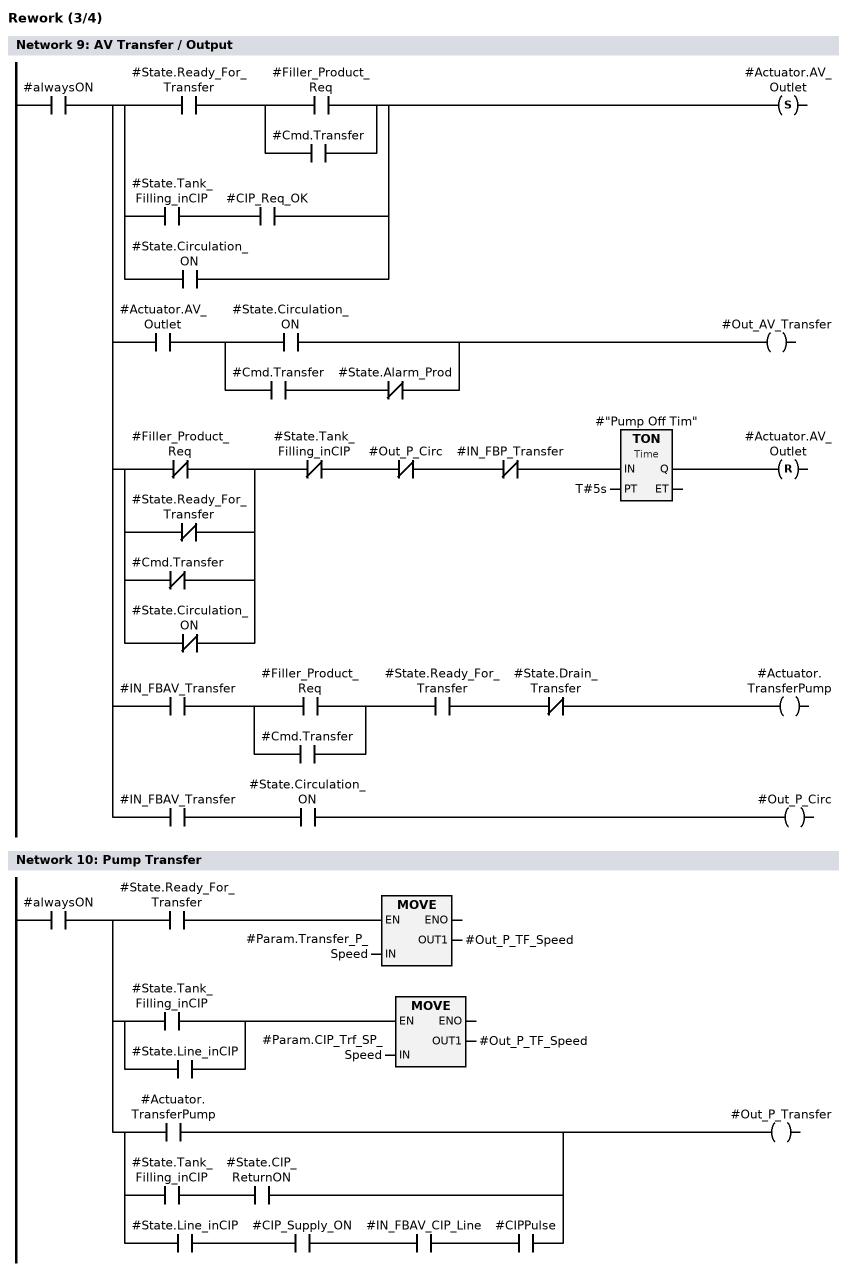
   RUNG wire#powerrail
      Contact( #alwaysON )
      wire#w1
      Contact( #State.Ready_For_Transfer )
      wire#w2
      Contact( #Filler_Product_Req )
      wire#w3
      S_Coil( #Actuator.AV_Outlet )
   END_RUNG
   RUNG wire#w2
      Contact( #Cmd.Transfer )
   END_RUNG wire#w3
   RUNG wire#w1
      Contact( #State.Tank_Filling_inCIP )
      Contact( #CIP_Req_OK )
   END_RUNG wire#w3
   RUNG wire#w1
      Contact( #State.Circulation_ON )
   END_RUNG wire#w3
   RUNG wire#w1
      Contact( #Actuator.AV_Outlet )
      wire#w4
      Contact( #State.Circulation_ON )
      wire#w5
      Coil( #Out_AV_Transfer )
   END_RUNG
   RUNG wire#w4
      Contact( #Cmd.Transfer )
      I_Contact( #State.Alarm_Prod )
   END_RUNG wire#w5
   RUNG wire#w1
      I_Contact( #Filler_Product_Req )
      wire#w6
      I_Contact( #State.Tank_Filling_inCIP )
      I_Contact( #Out_P_Circ )
      I_Contact( #IN_FBP_Transfer )
      { S7_Templates := "time_type := Time" } #"Pump Off Tim".TON(pt := T#5s, et =>)
      R_Coil( #Actuator.AV_Outlet )
   END_RUNG
   RUNG wire#w1
      I_Contact( #State.Ready_For_Transfer )
   END_RUNG wire#w6
   RUNG wire#w1
      I_Contact( #Cmd.Transfer )
   END_RUNG wire#w6
   RUNG wire#w1
      I_Contact( #State.Circulation_ON )
   END_RUNG wire#w6
   RUNG wire#w1
      Contact( #IN_FBAV_Transfer )
      wire#w7
      Contact( #Filler_Product_Req )
      wire#w8
      Contact( #State.Ready_For_Transfer )
      I_Contact( #State.Drain_Transfer )
      Coil( #Actuator.TransferPump )
   END_RUNG
   RUNG wire#w7
      Contact( #Cmd.Transfer )
   END_RUNG wire#w8
   RUNG wire#w1
      Contact( #IN_FBAV_Transfer )
      Contact( #State.Circulation_ON )
      Coil( #Out_P_Circ )
   END_RUNG
   // the same network as SCL:
   IF #alwaysON AND ((#State.Ready_For_Transfer AND (#Filler_Product_Req OR #Cmd.Transfer)) OR (#State.Tank_Filling_inCIP AND #CIP_Req_OK) OR #State.Circulation_ON) THEN
       #Actuator.AV_Outlet := TRUE;
   END_IF;
   #Out_AV_Transfer := #alwaysON AND #Actuator.AV_Outlet AND (#State.Circulation_ON OR (#Cmd.Transfer AND NOT #State.Alarm_Prod));
   #"Pump Off Tim"(IN := #alwaysON AND (NOT #Filler_Product_Req OR NOT #State.Ready_For_Transfer OR NOT #Cmd.Transfer OR NOT #State.Circulation_ON) AND NOT #State.Tank_Filling_inCIP AND NOT #Out_P_Circ AND NOT #IN_FBP_Transfer,   // TON
                   PT := T#5s);
   IF #"Pump Off Tim".Q THEN #Actuator.AV_Outlet := FALSE; END_IF;
   #Actuator.TransferPump := #alwaysON AND #IN_FBAV_Transfer AND (#Filler_Product_Req OR #Cmd.Transfer) AND #State.Ready_For_Transfer AND NOT #State.Drain_Transfer;
   #Out_P_Circ := #alwaysON AND #IN_FBAV_Transfer AND #State.Circulation_ON;
END_REGION

REGION Network 10: Pump Transfer
   RUNG wire#powerrail
      Contact( #alwaysON )
      wire#w1
      Contact( #State.Ready_For_Transfer )
      Move(in := #Param.Transfer_P_Speed, out1 => #Out_P_TF_Speed)
   END_RUNG
   RUNG wire#w1
      Contact( #State.Tank_Filling_inCIP )
      wire#w2
      Move(in := #Param.CIP_Trf_SP_Speed, out1 => #Out_P_TF_Speed)
   END_RUNG
   RUNG wire#w1
      Contact( #State.Line_inCIP )
   END_RUNG wire#w2
   RUNG wire#w1
      Contact( #Actuator.TransferPump )
      wire#w3
      Coil( #Out_P_Transfer )
   END_RUNG
   RUNG wire#w1
      Contact( #State.Tank_Filling_inCIP )
      Contact( #State.CIP_ReturnON )
   END_RUNG wire#w3
   RUNG wire#w1
      Contact( #State.Line_inCIP )
      Contact( #CIP_Supply_ON )
      Contact( #IN_FBAV_CIP_Line )
      Contact( #CIPPulse )
   END_RUNG wire#w3
   // the same network as SCL:
   IF #alwaysON AND #State.Ready_For_Transfer THEN #Out_P_TF_Speed := #Param.Transfer_P_Speed; END_IF;
   IF #alwaysON AND (#State.Tank_Filling_inCIP OR #State.Line_inCIP) THEN
       #Out_P_TF_Speed := #Param.CIP_Trf_SP_Speed;
   END_IF;
   #Out_P_Transfer := #alwaysON AND (#Actuator.TransferPump OR (#State.Tank_Filling_inCIP AND #State.CIP_ReturnON) OR (#State.Line_inCIP AND #CIP_Supply_ON AND #IN_FBAV_CIP_Line AND #CIPPulse));
END_REGION

REGION Network 11: State Transfer to FIlling
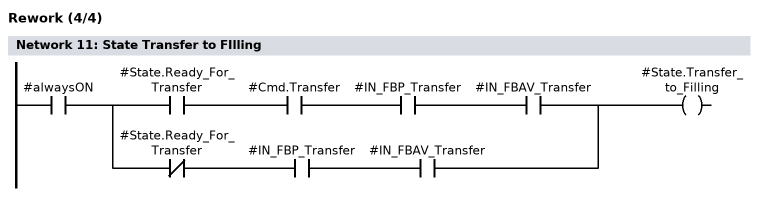
   RUNG wire#powerrail
      Contact( #alwaysON )
      wire#w1
      Contact( #State.Ready_For_Transfer )
      Contact( #Cmd.Transfer )
      Contact( #IN_FBP_Transfer )
      Contact( #IN_FBAV_Transfer )
      wire#w2
      Coil( #State.Transfer_to_Filling )
   END_RUNG
   RUNG wire#w1
      I_Contact( #State.Ready_For_Transfer )
      Contact( #IN_FBP_Transfer )
      Contact( #IN_FBAV_Transfer )
   END_RUNG wire#w2
   // the same network as SCL:
   #State.Transfer_to_Filling := #alwaysON AND ((#State.Ready_For_Transfer AND #Cmd.Transfer AND #IN_FBP_Transfer AND #IN_FBAV_Transfer) OR (NOT #State.Ready_For_Transfer AND #IN_FBP_Transfer AND #IN_FBAV_Transfer));
END_REGION
END_FUNCTION_BLOCK

FUNCTION_BLOCK "BFT_Type1"   // FB351, LAD
{ S7_Optimized_Access := 'TRUE' }
VERSION : 0.1
// Buffer Tank
// stored: AutoNumber false, IsIECCheckEnabled false, IsRetainMemResEnabled false, MemoryReserve 100, SetENOAutomatically false, UDAEnableTagReadback false
   VAR_INPUT
      "IN_FBAV.01" : Bool := FALSE;   // Tank Flushing Water Valve
      "IN_FBAV.02" : Bool := FALSE;   // Tank CIP Top Inlet Valve
      "IN_FBAV.03" : Bool := FALSE;   // Tank Tank Outlet Valve
      "IN_FBAV.04" : Bool := FALSE;   // Tank CIP Return Valve
      "IN_FBAV.05" : Bool := FALSE;   // Line CIP Bypass Valve
      "IN_FBAV.06" : Bool := FALSE;   // Tank Inlet Valve
      "IN_FBAV.07" : Bool := FALSE;   // Tank CIP Valve
      "IN_FBAV.08" : Bool := FALSE;   // Tank CIP Valve
      "IN_FBAV.09" : Bool := FALSE;   // Line CIP Valve
      IN_LT01 : Real;   // Tank Level Transmitter
      "IN_FBP.01" : Bool := FALSE;   // Transfer Pump
      "IN_P.01-Speed" : Real;   // Transfer Pump AV Speed
      "IN_FBP.02" : Bool := FALSE;   // CIP Pump
      "IN_P.02-Speed" : Real;   // CIP Pump AV Speed
      "IN_FBP.03" : Bool := FALSE;   // Supply Pump
      "IN_P.03-Speed" : Real;   // Supply Pump AV Speed
      DosePumpSpeed : Real;
      "DoseON-OFF" : Bool := FALSE;
      "DosePumpON-OFF" : Bool := FALSE;
      CIPPulse : Bool := FALSE;
      CIP_Supply_ON : Bool;
      LineTrf_OK : Bool := FALSE;
      LineFlush_OK : Bool;
      Loading_Busy : Bool;   // Other tank at loading
   END_VAR
   VAR_OUTPUT
      "OUT_AV.01" : Bool := FALSE;   // Tank Flushing Water Valve
      "OUT_AV.02" : Bool := FALSE;   // Tank CIP Top Inlet Valve
      "OUT_AV.03" : Bool := FALSE;   // Tank Tank Outlet Valve
      "OUT_AV.04" : Bool := FALSE;   // Tank CIP Return Valve
      "OUT_AV.05" : Bool := FALSE;   // Line CIP Bypass Valve
      "OUT_AV.06" : Bool := FALSE;   // Tank Inlet Valve
      "OUT_AV.07" : Bool := FALSE;   // Tank CIP Valve
      "OUT_AV.08" : Bool := FALSE;   // Tank CIP Valve
      "OUT_AV.09" : Bool := FALSE;   // Line CIP Valve
      "OUT_P.01" : Bool := FALSE;   // Transfer Pump
      "OUT_P.01-Speed" : Real;   // Transfer Pump AV Speed
      "OUT_P.02" : Bool := FALSE;   // CIP Pump
      "OUT_P.02-Speed" : Real;   // CIP Pump AV Speed
      "OUT_P.03" : Bool := FALSE;   // Supply Pump
      "OUT_P.03-Speed" : Real;   // Supply Pump AV Speed
      OUT_CIPTank_AVOpen : Bool;
      OUT_CIPLine_AVOpen : Bool;
   END_VAR
   VAR
      Cmd : Struct
         Inload : Bool;   // Start Loading
         Tank_CIP_Req : Bool;
         Line_CIP_Req : Bool;
         Flushing : Bool;   // Water Flushing
         RaadyForMix : Bool;   // Tank Ready for Blending
         Flush_Select : Byte;
      END_STRUCT;
      Param : Struct
         SP_Level_LL : Real := 10.0;
         SP_Level_ML : Real := 80.0;
         SP_Level_HL : Real := 100.0;
         SupplyPump_SP_Speed : Real := 80.0;
         L_Hi_Lim : Real := 100.0;
         L_Lo_Lim : Real := 0.0;
         L_Hys : Real := 5.0;
         FlushingTime : DInt := 10000;
         CIP_Trf_SP_Speed : Real := 80.0;
         CIP_Ret_ON_SP : Real := 5.0;
         CIP_Ret_OFF_SP : Real;
      END_STRUCT;
      State : Struct   // Tank in loading state
         Tank_inloading : Bool;
         Tank_inCIP : Bool;
         Line_inCIP : Bool;
         Flushing : Bool;
         Tank_LL : Bool;
         Tank_ML : Bool;
         Tank_HL : Bool;
         Inload_Enable : Bool;
         Tank_CIP_Enable : Bool;
         Line_CIP_Enable : Bool;
         Flushing_Enable : Bool;
         Flush_selected : Byte;
         CIP_Request_OK : Bool;
         CIP_ReturnON : Bool;
         Ready_For_Transfer_EN : Bool;   // Tank Ready for Transfer to Blending
         Ready_For_Transfer : Bool;   // Tank Ready for Transfer to Blending
         HWT_Status : Int;
         Transfer_to_Blend : Bool;
      END_STRUCT;
      alwaysON : Bool;
      L_Hys_Abs : Real;
      Hys_Level_HL : Real;
      Hys_Level_ML : Real;
      Hys_Level_LL : Real;
      r : Struct
         PosE1 : Bool;
         PosE2 : Bool;
         PosE3 : Bool;
         PosE4 : Bool;
         PosE5 : Bool;
         PosE6 : Bool;
         PosE7 : Bool;
         PosE8 : Bool;
         PosE9 : Bool;
         PosE10 : Bool;
         PosE11 : Bool;
         PosE12 : Bool;
         PosE13 : Bool;
         PosE14 : Bool;
         PosE15 : Bool;
         PosE16 : Bool;
         PosE17 : Bool;
         PosE18 : Bool;
         PosE19 : Bool;
         PosE20 : Bool;
         PosE21 : Bool;
         PosE22 : Bool;
         PosE23 : Bool;
         PosE24 : Bool;
         PosE25 : Bool;
         PosE26 : Bool;
         PosE27 : Bool;
         PosE28 : Bool;
         PosE29 : Bool;
         PosE30 : Bool;
         PosE31 : Bool;
         PosE32 : Bool;
      END_STRUCT;
      Actuator : Struct
         AV_Outlet : Bool;
         TransferPump : Bool;
         FlushPump : Bool;
         CV_Steam : Bool;
         Pump : Bool;
      END_STRUCT;
      FlushingTim : TON_TIME;
      SPumpTim { S7_SetPoint := 'True'} : TON_TIME;
      AVinloadTim { S7_SetPoint := 'True'} : TON_TIME;
   END_VAR
   VAR_TEMP   // added for the SCL form of the ladder/FBD networks
      _w1 : Bool;
      _w2 : Bool;
      _w3 : Bool;
      _w4 : Bool;
      _w5 : Bool;
      _w6 : Bool;
   END_VAR
BEGIN

REGION Network 1: Always_ON
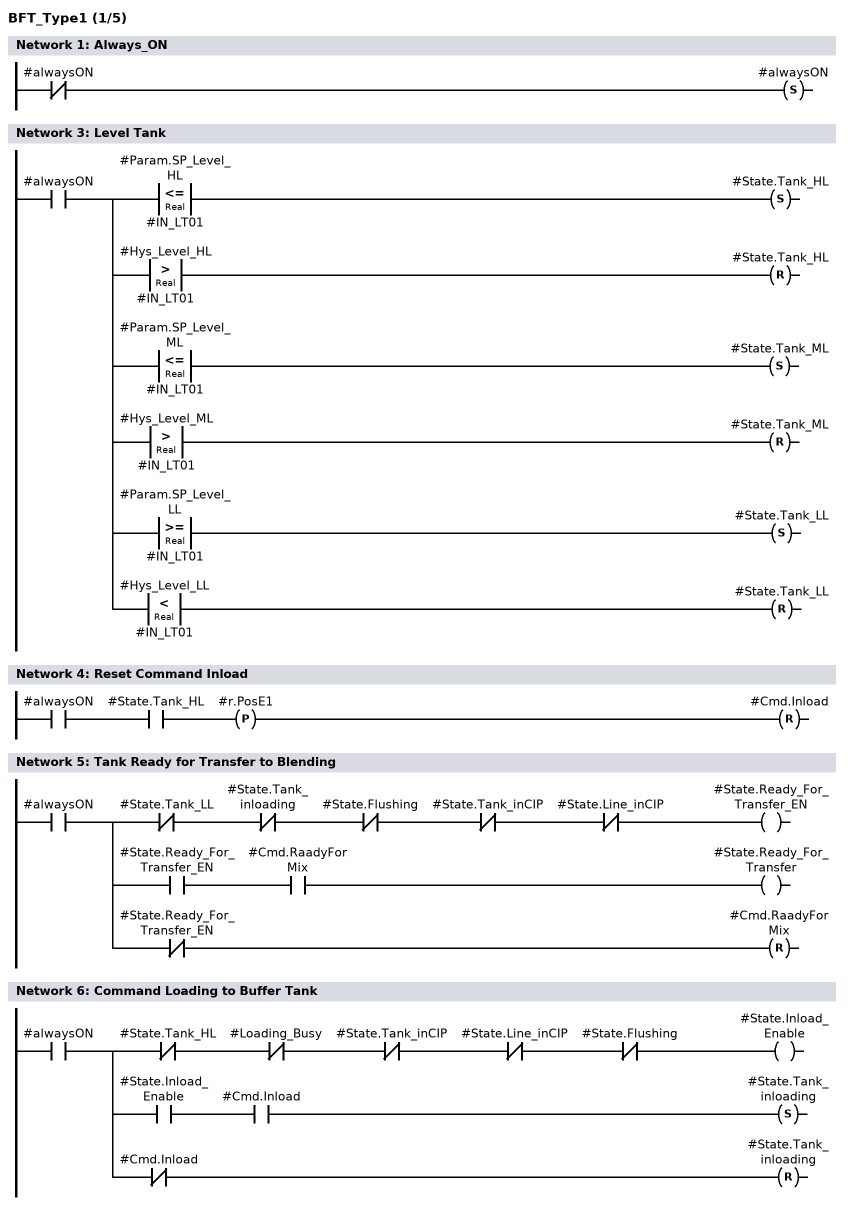
   RUNG wire#powerrail
      I_Contact( #alwaysON )
      S_Coil( #alwaysON )
   END_RUNG
   // the same network as SCL:
   IF NOT #alwaysON THEN #alwaysON := TRUE; END_IF;
END_REGION

NETWORK
TITLE = Hys Calculation
//Level Hys Absolute
      L     #Param.L_Hi_Lim;
      L     #Param.L_Lo_Lim;
      -R;
      L     100.0;
      /R;
      L     #Param.L_Hys;
      *R;
      T     #L_Hys_Abs;
//Tank High Level
      L     #Param.SP_Level_HL;
      L     #L_Hys_Abs;
      -R;
      T     #Hys_Level_HL;
//Tank Mid Level
      L     #Param.SP_Level_ML;
      L     #L_Hys_Abs;
      -R;
      T     #Hys_Level_ML;
//Tank Low Level
      L     #Param.SP_Level_LL;
      L     #L_Hys_Abs;
      +R;
      T     #Hys_Level_LL;


REGION Network 3: Level Tank
   RUNG wire#powerrail
      Contact( #alwaysON )
      wire#w1
      { S7_Templates := "SrcType := Real" } LE_Contact(in1 := #Param.SP_Level_HL, in2 := #IN_LT01)
      S_Coil( #State.Tank_HL )
   END_RUNG
   RUNG wire#w1
      { S7_Templates := "SrcType := Real" } GT_Contact(in1 := #Hys_Level_HL, in2 := #IN_LT01)
      R_Coil( #State.Tank_HL )
   END_RUNG
   RUNG wire#w1
      { S7_Templates := "SrcType := Real" } LE_Contact(in1 := #Param.SP_Level_ML, in2 := #IN_LT01)
      S_Coil( #State.Tank_ML )
   END_RUNG
   RUNG wire#w1
      { S7_Templates := "SrcType := Real" } GT_Contact(in1 := #Hys_Level_ML, in2 := #IN_LT01)
      R_Coil( #State.Tank_ML )
   END_RUNG
   RUNG wire#w1
      { S7_Templates := "SrcType := Real" } GE_Contact(in1 := #Param.SP_Level_LL, in2 := #IN_LT01)
      S_Coil( #State.Tank_LL )
   END_RUNG
   RUNG wire#w1
      { S7_Templates := "SrcType := Real" } LT_Contact(in1 := #Hys_Level_LL, in2 := #IN_LT01)
      R_Coil( #State.Tank_LL )
   END_RUNG
   // the same network as SCL:
   IF #alwaysON AND (#Param.SP_Level_HL <= #IN_LT01) THEN #State.Tank_HL := TRUE; END_IF;
   IF #alwaysON AND (#Hys_Level_HL > #IN_LT01) THEN #State.Tank_HL := FALSE; END_IF;
   IF #alwaysON AND (#Param.SP_Level_ML <= #IN_LT01) THEN #State.Tank_ML := TRUE; END_IF;
   IF #alwaysON AND (#Hys_Level_ML > #IN_LT01) THEN #State.Tank_ML := FALSE; END_IF;
   IF #alwaysON AND (#Param.SP_Level_LL >= #IN_LT01) THEN #State.Tank_LL := TRUE; END_IF;
   IF #alwaysON AND (#Hys_Level_LL < #IN_LT01) THEN #State.Tank_LL := FALSE; END_IF;
END_REGION

REGION Network 4: Reset Command Inload
   RUNG wire#powerrail
      Contact( #alwaysON )
      Contact( #State.Tank_HL )
      P_Trig( #r.PosE1 )
      R_Coil( #Cmd.Inload )
   END_RUNG
   // the same network as SCL:
   #_w1 := #alwaysON AND #State.Tank_HL;
   #_w2 := #_w1 AND NOT #r.PosE1;   // rising edge
   #r.PosE1 := #_w1;
   IF #_w2 THEN #Cmd.Inload := FALSE; END_IF;
END_REGION

REGION Network 5: Tank Ready for Transfer to Blending
   RUNG wire#powerrail
      Contact( #alwaysON )
      wire#w1
      I_Contact( #State.Tank_LL )
      I_Contact( #State.Tank_inloading )
      I_Contact( #State.Flushing )
      I_Contact( #State.Tank_inCIP )
      I_Contact( #State.Line_inCIP )
      Coil( #State.Ready_For_Transfer_EN )
   END_RUNG
   RUNG wire#w1
      Contact( #State.Ready_For_Transfer_EN )
      Contact( #Cmd.RaadyForMix )
      Coil( #State.Ready_For_Transfer )
   END_RUNG
   RUNG wire#w1
      I_Contact( #State.Ready_For_Transfer_EN )
      R_Coil( #Cmd.RaadyForMix )
   END_RUNG
   // the same network as SCL:
   #State.Ready_For_Transfer_EN := #alwaysON AND NOT #State.Tank_LL AND NOT #State.Tank_inloading AND NOT #State.Flushing AND NOT #State.Tank_inCIP AND NOT #State.Line_inCIP;
   #State.Ready_For_Transfer := #alwaysON AND #State.Ready_For_Transfer_EN AND #Cmd.RaadyForMix;
   IF #alwaysON AND NOT #State.Ready_For_Transfer_EN THEN #Cmd.RaadyForMix := FALSE; END_IF;
END_REGION

REGION Network 6: Command Loading to Buffer Tank
   RUNG wire#powerrail
      Contact( #alwaysON )
      wire#w1
      I_Contact( #State.Tank_HL )
      I_Contact( #Loading_Busy )
      I_Contact( #State.Tank_inCIP )
      I_Contact( #State.Line_inCIP )
      I_Contact( #State.Flushing )
      Coil( #State.Inload_Enable )
   END_RUNG
   RUNG wire#w1
      Contact( #State.Inload_Enable )
      Contact( #Cmd.Inload )
      S_Coil( #State.Tank_inloading )
   END_RUNG
   RUNG wire#w1
      I_Contact( #Cmd.Inload )
      R_Coil( #State.Tank_inloading )
   END_RUNG
   // the same network as SCL:
   #State.Inload_Enable := #alwaysON AND NOT #State.Tank_HL AND NOT #Loading_Busy AND NOT #State.Tank_inCIP AND NOT #State.Line_inCIP AND NOT #State.Flushing;
   IF #alwaysON AND #State.Inload_Enable AND #Cmd.Inload THEN #State.Tank_inloading := TRUE; END_IF;
   IF #alwaysON AND NOT #Cmd.Inload THEN #State.Tank_inloading := FALSE; END_IF;
END_REGION

REGION Network 7: Choose Flush Destination
   // #Cmd.Flush_Select.%X0 = T-20.00
   // #Cmd.Flush_Select.%X1 = T-21.00
   // #Cmd.Flush_Select.%X2 = T-30.00
   // #Cmd.Flush_Select.%X3 = T-31.00
   // #Cmd.Flush_Select.%X4 = Drain
   // #Cmd.Flush_Select.%X5 = Flush_Selected
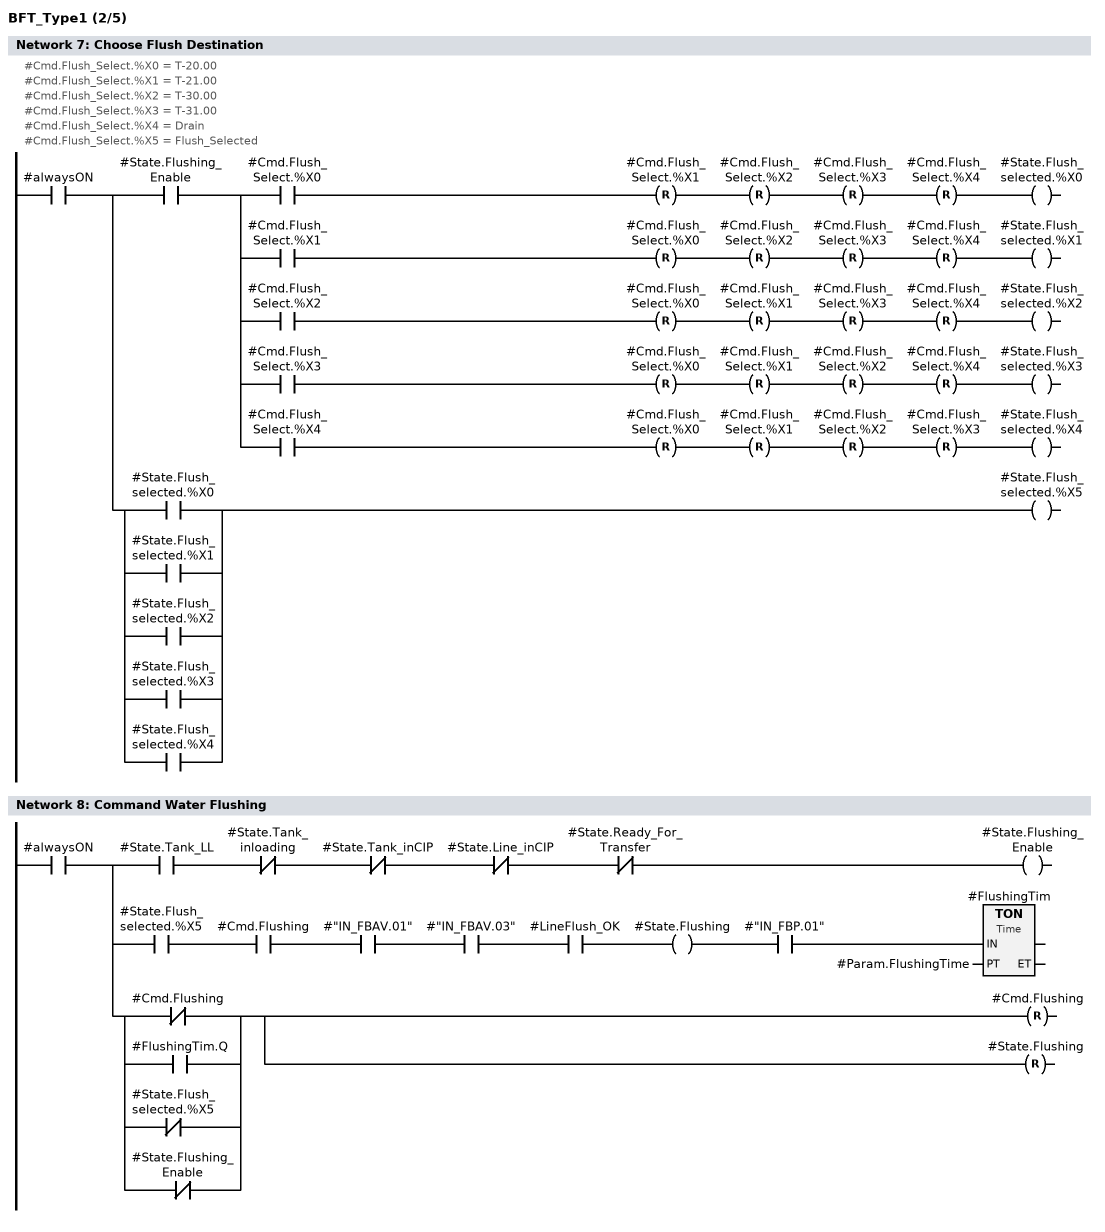
   RUNG wire#powerrail
      Contact( #alwaysON )
      wire#w1
      Contact( #State.Flushing_Enable )
      wire#w2
      Contact( #Cmd.Flush_Select.%X0 )
      R_Coil( #Cmd.Flush_Select.%X1 )
      R_Coil( #Cmd.Flush_Select.%X2 )
      R_Coil( #Cmd.Flush_Select.%X3 )
      R_Coil( #Cmd.Flush_Select.%X4 )
      Coil( #State.Flush_selected.%X0 )
   END_RUNG
   RUNG wire#w2
      Contact( #Cmd.Flush_Select.%X1 )
      R_Coil( #Cmd.Flush_Select.%X0 )
      R_Coil( #Cmd.Flush_Select.%X2 )
      R_Coil( #Cmd.Flush_Select.%X3 )
      R_Coil( #Cmd.Flush_Select.%X4 )
      Coil( #State.Flush_selected.%X1 )
   END_RUNG
   RUNG wire#w2
      Contact( #Cmd.Flush_Select.%X2 )
      R_Coil( #Cmd.Flush_Select.%X0 )
      R_Coil( #Cmd.Flush_Select.%X1 )
      R_Coil( #Cmd.Flush_Select.%X3 )
      R_Coil( #Cmd.Flush_Select.%X4 )
      Coil( #State.Flush_selected.%X2 )
   END_RUNG
   RUNG wire#w2
      Contact( #Cmd.Flush_Select.%X3 )
      R_Coil( #Cmd.Flush_Select.%X0 )
      R_Coil( #Cmd.Flush_Select.%X1 )
      R_Coil( #Cmd.Flush_Select.%X2 )
      R_Coil( #Cmd.Flush_Select.%X4 )
      Coil( #State.Flush_selected.%X3 )
   END_RUNG
   RUNG wire#w2
      Contact( #Cmd.Flush_Select.%X4 )
      R_Coil( #Cmd.Flush_Select.%X0 )
      R_Coil( #Cmd.Flush_Select.%X1 )
      R_Coil( #Cmd.Flush_Select.%X2 )
      R_Coil( #Cmd.Flush_Select.%X3 )
      Coil( #State.Flush_selected.%X4 )
   END_RUNG
   RUNG wire#w1
      Contact( #State.Flush_selected.%X0 )
      wire#w3
      Coil( #State.Flush_selected.%X5 )
   END_RUNG
   RUNG wire#w1
      Contact( #State.Flush_selected.%X1 )
   END_RUNG wire#w3
   RUNG wire#w1
      Contact( #State.Flush_selected.%X2 )
   END_RUNG wire#w3
   RUNG wire#w1
      Contact( #State.Flush_selected.%X3 )
   END_RUNG wire#w3
   RUNG wire#w1
      Contact( #State.Flush_selected.%X4 )
   END_RUNG wire#w3
   // the same network as SCL:
   #_w1 := #alwaysON AND #State.Flushing_Enable;
   #_w2 := #_w1 AND #Cmd.Flush_Select.%X0;
   IF #_w2 THEN
       #Cmd.Flush_Select.%X1 := FALSE;
       #Cmd.Flush_Select.%X2 := FALSE;
       #Cmd.Flush_Select.%X3 := FALSE;
       #Cmd.Flush_Select.%X4 := FALSE;
   END_IF;
   #State.Flush_selected.%X0 := #_w2;
   #_w3 := #_w1 AND #Cmd.Flush_Select.%X1;
   IF #_w3 THEN
       #Cmd.Flush_Select.%X0 := FALSE;
       #Cmd.Flush_Select.%X2 := FALSE;
       #Cmd.Flush_Select.%X3 := FALSE;
       #Cmd.Flush_Select.%X4 := FALSE;
   END_IF;
   #State.Flush_selected.%X1 := #_w3;
   #_w4 := #_w1 AND #Cmd.Flush_Select.%X2;
   IF #_w4 THEN
       #Cmd.Flush_Select.%X0 := FALSE;
       #Cmd.Flush_Select.%X1 := FALSE;
       #Cmd.Flush_Select.%X3 := FALSE;
       #Cmd.Flush_Select.%X4 := FALSE;
   END_IF;
   #State.Flush_selected.%X2 := #_w4;
   #_w5 := #_w1 AND #Cmd.Flush_Select.%X3;
   IF #_w5 THEN
       #Cmd.Flush_Select.%X0 := FALSE;
       #Cmd.Flush_Select.%X1 := FALSE;
       #Cmd.Flush_Select.%X2 := FALSE;
       #Cmd.Flush_Select.%X4 := FALSE;
   END_IF;
   #State.Flush_selected.%X3 := #_w5;
   #_w6 := #_w1 AND #Cmd.Flush_Select.%X4;
   IF #_w6 THEN
       #Cmd.Flush_Select.%X0 := FALSE;
       #Cmd.Flush_Select.%X1 := FALSE;
       #Cmd.Flush_Select.%X2 := FALSE;
       #Cmd.Flush_Select.%X3 := FALSE;
   END_IF;
   #State.Flush_selected.%X4 := #_w6;
   #State.Flush_selected.%X5 := #alwaysON AND (#State.Flush_selected.%X0 OR #State.Flush_selected.%X1 OR #State.Flush_selected.%X2 OR #State.Flush_selected.%X3 OR #State.Flush_selected.%X4);
END_REGION

REGION Network 8: Command Water Flushing
   RUNG wire#powerrail
      Contact( #alwaysON )
      wire#w1
      Contact( #State.Tank_LL )
      I_Contact( #State.Tank_inloading )
      I_Contact( #State.Tank_inCIP )
      I_Contact( #State.Line_inCIP )
      I_Contact( #State.Ready_For_Transfer )
      Coil( #State.Flushing_Enable )
   END_RUNG
   RUNG wire#w1
      Contact( #State.Flush_selected.%X5 )
      Contact( #Cmd.Flushing )
      Contact( #"IN_FBAV.01" )
      Contact( #"IN_FBAV.03" )
      Contact( #LineFlush_OK )
      Coil( #State.Flushing )
      Contact( #"IN_FBP.01" )
      { S7_Templates := "time_type := Time" } #FlushingTim.TON(pt := #Param.FlushingTime, et =>)
   END_RUNG
   RUNG wire#w1
      I_Contact( #Cmd.Flushing )
      wire#w2
      R_Coil( #Cmd.Flushing )
   END_RUNG
   RUNG wire#w1
      Contact( #FlushingTim.Q )
   END_RUNG wire#w2
   RUNG wire#w1
      I_Contact( #State.Flush_selected.%X5 )
   END_RUNG wire#w2
   RUNG wire#w1
      I_Contact( #State.Flushing_Enable )
   END_RUNG wire#w2
   RUNG wire#w2
      R_Coil( #State.Flushing )
   END_RUNG
   // the same network as SCL:
   #State.Flushing_Enable := #alwaysON AND #State.Tank_LL AND NOT #State.Tank_inloading AND NOT #State.Tank_inCIP AND NOT #State.Line_inCIP AND NOT #State.Ready_For_Transfer;
   #State.Flushing := #alwaysON AND #State.Flush_selected.%X5 AND #Cmd.Flushing AND #"IN_FBAV.01" AND #"IN_FBAV.03" AND #LineFlush_OK;
   #FlushingTim(IN := #State.Flushing AND #"IN_FBP.01", PT := #Param.FlushingTime);   // TON
   #_w1 := #alwaysON AND (NOT #Cmd.Flushing OR #FlushingTim.Q OR NOT #State.Flush_selected.%X5 OR NOT #State.Flushing_Enable);
   IF #_w1 THEN
       #Cmd.Flushing := FALSE;
       #State.Flushing := FALSE;
   END_IF;
END_REGION

REGION Network 9: Flushing Destination AV and Pump
   // #Cmd.Flush_Select.%X0 = T-20.00
   // #Cmd.Flush_Select.%X1 = T-21.00
   // #Cmd.Flush_Select.%X2 = T-30.00
   // #Cmd.Flush_Select.%X3 = T-31.00
   // #Cmd.Flush_Select.%X4 = Drain
   // #Cmd.Flush_Select.%X5 = Flush_Selected
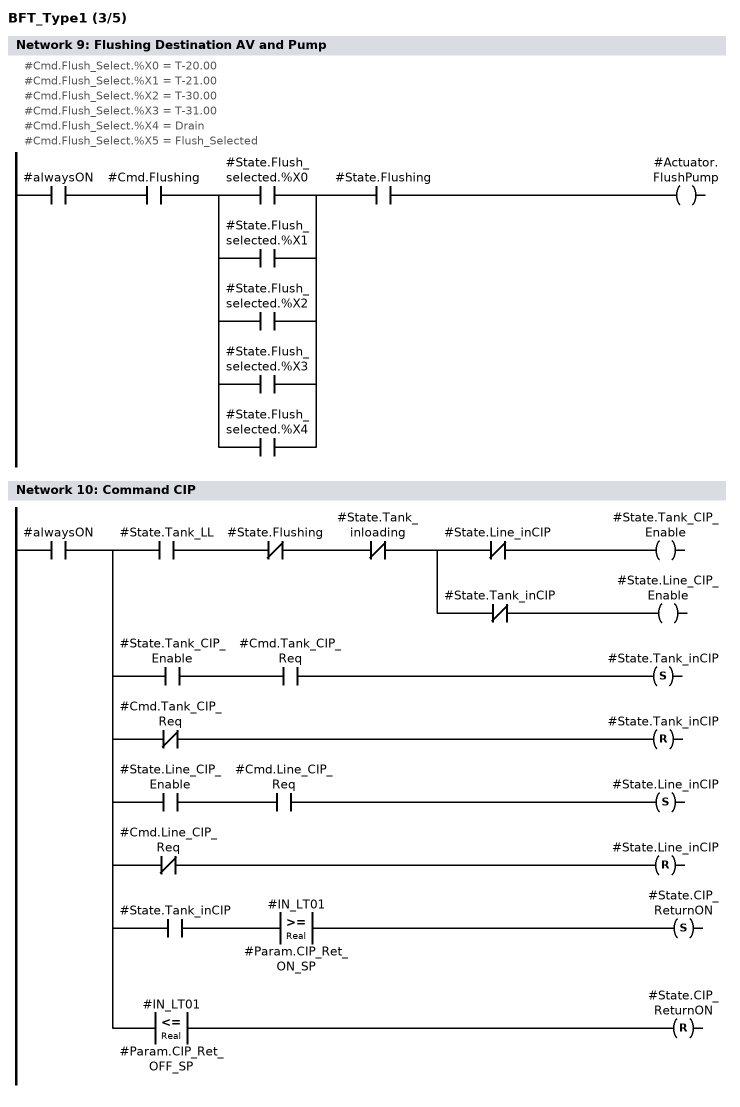
   RUNG wire#powerrail
      Contact( #alwaysON )
      Contact( #Cmd.Flushing )
      wire#w1
      Contact( #State.Flush_selected.%X0 )
      wire#w2
      Contact( #State.Flushing )
      Coil( #Actuator.FlushPump )
   END_RUNG
   RUNG wire#w1
      Contact( #State.Flush_selected.%X1 )
   END_RUNG wire#w2
   RUNG wire#w1
      Contact( #State.Flush_selected.%X2 )
   END_RUNG wire#w2
   RUNG wire#w1
      Contact( #State.Flush_selected.%X3 )
   END_RUNG wire#w2
   RUNG wire#w1
      Contact( #State.Flush_selected.%X4 )
   END_RUNG wire#w2
   // the same network as SCL:
   #Actuator.FlushPump := #alwaysON AND #Cmd.Flushing AND (#State.Flush_selected.%X0 OR #State.Flush_selected.%X1 OR #State.Flush_selected.%X2 OR #State.Flush_selected.%X3 OR #State.Flush_selected.%X4) AND #State.Flushing;
END_REGION

REGION Network 10: Command CIP
   RUNG wire#powerrail
      Contact( #alwaysON )
      wire#w1
      Contact( #State.Tank_LL )
      I_Contact( #State.Flushing )
      I_Contact( #State.Tank_inloading )
      wire#w2
      I_Contact( #State.Line_inCIP )
      Coil( #State.Tank_CIP_Enable )
   END_RUNG
   RUNG wire#w2
      I_Contact( #State.Tank_inCIP )
      Coil( #State.Line_CIP_Enable )
   END_RUNG
   RUNG wire#w1
      Contact( #State.Tank_CIP_Enable )
      Contact( #Cmd.Tank_CIP_Req )
      S_Coil( #State.Tank_inCIP )
   END_RUNG
   RUNG wire#w1
      I_Contact( #Cmd.Tank_CIP_Req )
      R_Coil( #State.Tank_inCIP )
   END_RUNG
   RUNG wire#w1
      Contact( #State.Line_CIP_Enable )
      Contact( #Cmd.Line_CIP_Req )
      S_Coil( #State.Line_inCIP )
   END_RUNG
   RUNG wire#w1
      I_Contact( #Cmd.Line_CIP_Req )
      R_Coil( #State.Line_inCIP )
   END_RUNG
   RUNG wire#w1
      Contact( #State.Tank_inCIP )
      { S7_Templates := "SrcType := Real" } GE_Contact(in1 := #IN_LT01, in2 := #Param.CIP_Ret_ON_SP)
      S_Coil( #State.CIP_ReturnON )
   END_RUNG
   RUNG wire#w1
      { S7_Templates := "SrcType := Real" } LE_Contact(in1 := #IN_LT01, in2 := #Param.CIP_Ret_OFF_SP)
      R_Coil( #State.CIP_ReturnON )
   END_RUNG
   // the same network as SCL:
   #_w1 := #alwaysON AND #State.Tank_LL AND NOT #State.Flushing AND NOT #State.Tank_inloading;
   #State.Tank_CIP_Enable := #_w1 AND NOT #State.Line_inCIP;
   #State.Line_CIP_Enable := #_w1 AND NOT #State.Tank_inCIP;
   IF #alwaysON AND #State.Tank_CIP_Enable AND #Cmd.Tank_CIP_Req THEN #State.Tank_inCIP := TRUE; END_IF;
   IF #alwaysON AND NOT #Cmd.Tank_CIP_Req THEN #State.Tank_inCIP := FALSE; END_IF;
   IF #alwaysON AND #State.Line_CIP_Enable AND #Cmd.Line_CIP_Req THEN #State.Line_inCIP := TRUE; END_IF;
   IF #alwaysON AND NOT #Cmd.Line_CIP_Req THEN #State.Line_inCIP := FALSE; END_IF;
   IF #alwaysON AND #State.Tank_inCIP AND (#IN_LT01 >= #Param.CIP_Ret_ON_SP) THEN
       #State.CIP_ReturnON := TRUE;
   END_IF;
   IF #alwaysON AND (#IN_LT01 <= #Param.CIP_Ret_OFF_SP) THEN #State.CIP_ReturnON := FALSE; END_IF;
END_REGION

REGION Network 11: Loading AV and Pump
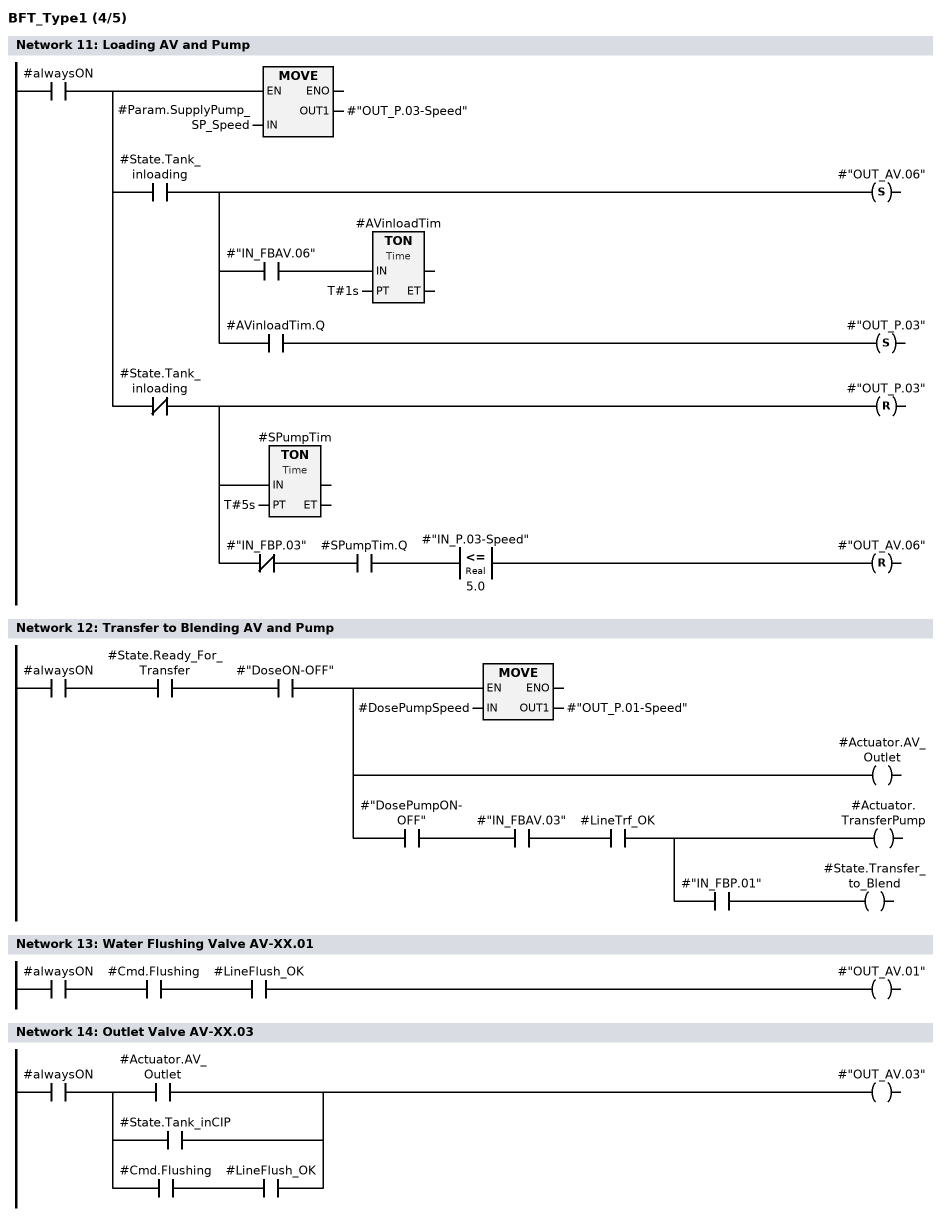
   RUNG wire#powerrail
      Contact( #alwaysON )
      wire#w1
      Move(in := #Param.SupplyPump_SP_Speed, out1 => #"OUT_P.03-Speed")
   END_RUNG
   RUNG wire#w1
      Contact( #State.Tank_inloading )
      wire#w2
      S_Coil( #"OUT_AV.06" )
   END_RUNG
   RUNG wire#w2
      Contact( #"IN_FBAV.06" )
      { S7_Templates := "time_type := Time" } #AVinloadTim.TON(pt := T#1s, et =>)
   END_RUNG
   RUNG wire#w2
      Contact( #AVinloadTim.Q )
      S_Coil( #"OUT_P.03" )
   END_RUNG
   RUNG wire#w1
      I_Contact( #State.Tank_inloading )
      wire#w3
      R_Coil( #"OUT_P.03" )
   END_RUNG
   RUNG wire#w3
      { S7_Templates := "time_type := Time" } #SPumpTim.TON(pt := T#5s, et =>)
   END_RUNG
   RUNG wire#w3
      I_Contact( #"IN_FBP.03" )
      Contact( #SPumpTim.Q )
      { S7_Templates := "SrcType := Real" } LE_Contact(in1 := #"IN_P.03-Speed", in2 := 5.0)
      R_Coil( #"OUT_AV.06" )
   END_RUNG
   // the same network as SCL:
   IF #alwaysON THEN #"OUT_P.03-Speed" := #Param.SupplyPump_SP_Speed; END_IF;
   #_w1 := #alwaysON AND #State.Tank_inloading;
   IF #_w1 THEN #"OUT_AV.06" := TRUE; END_IF;
   #AVinloadTim(IN := #_w1 AND #"IN_FBAV.06", PT := T#1s);   // TON
   IF #_w1 AND #AVinloadTim.Q THEN #"OUT_P.03" := TRUE; END_IF;
   #_w2 := #alwaysON AND NOT #State.Tank_inloading;
   IF #_w2 THEN #"OUT_P.03" := FALSE; END_IF;
   #SPumpTim(IN := #_w2, PT := T#5s);   // TON
   IF #_w2 AND NOT #"IN_FBP.03" AND #SPumpTim.Q AND (#"IN_P.03-Speed" <= 5.0) THEN
       #"OUT_AV.06" := FALSE;
   END_IF;
END_REGION

REGION Network 12: Transfer to Blending AV and Pump
   RUNG wire#powerrail
      Contact( #alwaysON )
      Contact( #State.Ready_For_Transfer )
      Contact( #"DoseON-OFF" )
      wire#w1
      Move(in := #DosePumpSpeed, out1 => #"OUT_P.01-Speed")
   END_RUNG
   RUNG wire#w1
      Coil( #Actuator.AV_Outlet )
   END_RUNG
   RUNG wire#w1
      Contact( #"DosePumpON-OFF" )
      Contact( #"IN_FBAV.03" )
      Contact( #LineTrf_OK )
      wire#w2
      Coil( #Actuator.TransferPump )
   END_RUNG
   RUNG wire#w2
      Contact( #"IN_FBP.01" )
      Coil( #State.Transfer_to_Blend )
   END_RUNG
   // the same network as SCL:
   #_w1 := #alwaysON AND #State.Ready_For_Transfer AND #"DoseON-OFF";
   IF #_w1 THEN #"OUT_P.01-Speed" := #DosePumpSpeed; END_IF;
   #Actuator.AV_Outlet := #_w1;
   #Actuator.TransferPump := #_w1 AND #"DosePumpON-OFF" AND #"IN_FBAV.03" AND #LineTrf_OK;
   #State.Transfer_to_Blend := #Actuator.TransferPump AND #"IN_FBP.01";
END_REGION

REGION Network 13: Water Flushing Valve AV-XX.01
   RUNG wire#powerrail
      Contact( #alwaysON )
      Contact( #Cmd.Flushing )
      Contact( #LineFlush_OK )
      Coil( #"OUT_AV.01" )
   END_RUNG
   // the same network as SCL:
   #"OUT_AV.01" := #alwaysON AND #Cmd.Flushing AND #LineFlush_OK;
END_REGION

REGION Network 14: Outlet Valve AV-XX.03
   RUNG wire#powerrail
      Contact( #alwaysON )
      wire#w1
      Contact( #Actuator.AV_Outlet )
      wire#w2
      Coil( #"OUT_AV.03" )
   END_RUNG
   RUNG wire#w1
      Contact( #State.Tank_inCIP )
   END_RUNG wire#w2
   RUNG wire#w1
      Contact( #Cmd.Flushing )
      Contact( #LineFlush_OK )
   END_RUNG wire#w2
   // the same network as SCL:
   #"OUT_AV.03" := #alwaysON AND (#Actuator.AV_Outlet OR #State.Tank_inCIP OR (#Cmd.Flushing AND #LineFlush_OK));
END_REGION

REGION Network 15: CIP Valve AV-XX.02, 04, 07
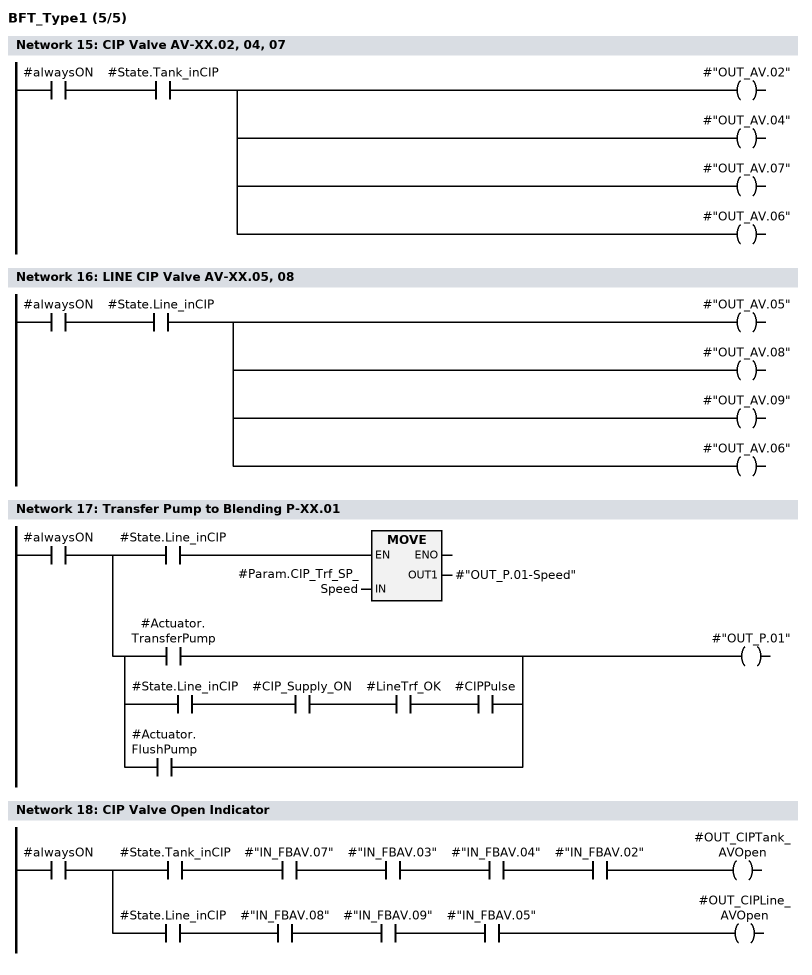
   RUNG wire#powerrail
      Contact( #alwaysON )
      Contact( #State.Tank_inCIP )
      wire#w1
      Coil( #"OUT_AV.02" )
   END_RUNG
   RUNG wire#w1
      Coil( #"OUT_AV.04" )
   END_RUNG
   RUNG wire#w1
      Coil( #"OUT_AV.07" )
   END_RUNG
   RUNG wire#w1
      Coil( #"OUT_AV.06" )
   END_RUNG
   // the same network as SCL:
   #"OUT_AV.02" := #alwaysON AND #State.Tank_inCIP;
   #"OUT_AV.04" := #"OUT_AV.02";
   #"OUT_AV.07" := #"OUT_AV.02";
   #"OUT_AV.06" := #"OUT_AV.02";
END_REGION

REGION Network 16: LINE CIP Valve AV-XX.05, 08
   RUNG wire#powerrail
      Contact( #alwaysON )
      Contact( #State.Line_inCIP )
      wire#w1
      Coil( #"OUT_AV.05" )
   END_RUNG
   RUNG wire#w1
      Coil( #"OUT_AV.08" )
   END_RUNG
   RUNG wire#w1
      Coil( #"OUT_AV.09" )
   END_RUNG
   RUNG wire#w1
      Coil( #"OUT_AV.06" )
   END_RUNG
   // the same network as SCL:
   #"OUT_AV.05" := #alwaysON AND #State.Line_inCIP;
   #"OUT_AV.08" := #"OUT_AV.05";
   #"OUT_AV.09" := #"OUT_AV.05";
   #"OUT_AV.06" := #"OUT_AV.05";
END_REGION

REGION Network 17: Transfer Pump to Blending P-XX.01
   RUNG wire#powerrail
      Contact( #alwaysON )
      wire#w1
      Contact( #State.Line_inCIP )
      Move(in := #Param.CIP_Trf_SP_Speed, out1 => #"OUT_P.01-Speed")
   END_RUNG
   RUNG wire#w1
      Contact( #Actuator.TransferPump )
      wire#w2
      Coil( #"OUT_P.01" )
   END_RUNG
   RUNG wire#w1
      Contact( #State.Line_inCIP )
      Contact( #CIP_Supply_ON )
      Contact( #LineTrf_OK )
      Contact( #CIPPulse )
   END_RUNG wire#w2
   RUNG wire#w1
      Contact( #Actuator.FlushPump )
   END_RUNG wire#w2
   // the same network as SCL:
   IF #alwaysON AND #State.Line_inCIP THEN #"OUT_P.01-Speed" := #Param.CIP_Trf_SP_Speed; END_IF;
   #"OUT_P.01" := #alwaysON AND (#Actuator.TransferPump OR (#State.Line_inCIP AND #CIP_Supply_ON AND #LineTrf_OK AND #CIPPulse) OR #Actuator.FlushPump);
END_REGION

REGION Network 18: CIP Valve Open Indicator
   RUNG wire#powerrail
      Contact( #alwaysON )
      wire#w1
      Contact( #State.Tank_inCIP )
      Contact( #"IN_FBAV.07" )
      Contact( #"IN_FBAV.03" )
      Contact( #"IN_FBAV.04" )
      Contact( #"IN_FBAV.02" )
      Coil( #OUT_CIPTank_AVOpen )
   END_RUNG
   RUNG wire#w1
      Contact( #State.Line_inCIP )
      Contact( #"IN_FBAV.08" )
      Contact( #"IN_FBAV.09" )
      Contact( #"IN_FBAV.05" )
      Coil( #OUT_CIPLine_AVOpen )
   END_RUNG
   // the same network as SCL:
   #OUT_CIPTank_AVOpen := #alwaysON AND #State.Tank_inCIP AND #"IN_FBAV.07" AND #"IN_FBAV.03" AND #"IN_FBAV.04" AND #"IN_FBAV.02";
   #OUT_CIPLine_AVOpen := #alwaysON AND #State.Line_inCIP AND #"IN_FBAV.08" AND #"IN_FBAV.09" AND #"IN_FBAV.05";
END_REGION
END_FUNCTION_BLOCK

FUNCTION_BLOCK "Analogue"
TITLE = Analogue
{ S7_Optimized_Access := 'FALSE' }
AUTHOR : RM
FAMILY : MON
VERSION : 0.1
   VAR_INPUT 
      LOCK : Bool;
      ERR_EXTERN : Bool;
      LIOP_SEL : Bool;
      L_SIM : Bool;
      L_RESET : Bool;
      IN_MODE : Bool;
      BIPOLAR : Bool;
      IN_INT : Int := 0;
      IN : Real := 55.0;
      IN_SIM : Real := 55.0;
      HI_LIM : Real := 100.0;
      LO_LIM : Real;
      LIM_ULA_Enable : Bool;
      LIM_ULA : Real := 90.0;
      LIM_ULW_Enable : Bool;
      LIM_ULW : Real := 80.0;
      LIM_LLW_Enable : Bool;
      LIM_LLW : Real := 20.0;
      LIM_LLA_Enable : Bool;
      LIM_LLA : Real := 10.0;
      LIM_HYS_Set : Bool;
      LIM_HYS : Real;
      INSTANCE : String := 'Analogue_001';
      RESTART : Bool;
   END_VAR

   VAR_OUTPUT 
      QdwState : DWord;
      QOUT : Real;
      QHI_LIM : Real;
      QLO_LIM : Real;
      QLIM_ULA_Enable : Bool;
      QLIM_ULA : Real;
      QLIM_ULW_Enable : Bool;
      QLIM_ULW : Real;
      QLIM_LLW_Enable : Bool;
      QLIM_LLW : Real;
      QLIM_LLA_Enable : Bool;
      QLIM_LLA : Real;
      QLIM_HYS : Real;
      QALARM_UL : Bool;
      QWARN_UL : Bool;
      QWARN_LL : Bool;
      QALARM_LL : Bool;
      QSIM : Bool;
      QLOCK : Bool;
      QERR : Bool;
      QERR_EXT : Bool;
      QERR_OVERRUN : Bool;
      QERR_HIGHRANGE : Bool;
      QERR_LOWRANGE : Bool;
      QERR_WIRE : Bool;
      QwAlarm : Word;
   END_VAR

   VAR_IN_OUT 
      VISIBILITY : Byte := 0;
      OPdwCmd : DWord;
   END_VAR

   VAR 
      OP_RESET : Bool;
      QLIM_HYS_Set : Bool;
      QIN_MODE : Bool;
      OP_LIM_ULA : Real;
      OP_LIM_ULW : Real;
      OP_LIM_LLW : Real;
      OP_LIM_LLA : Real;
      OP_SIM_Value : Real;
      OP_LIM_HYS_Perc : Real;
      OP_LIM_HYS_Abs : Real;
      OP_HI_LIM : Real;
      OP_LO_LIM : Real;
      OP_VISIBILITY : Byte;
      VISIBILITY_OLD : Byte;
      SEF_L_RESET_Link : Bool;
      Condition_SEF_L_RESET_Link : Bool;
      SEF_L_RESET_OP : Bool;
      Condition_Enable_ULA : Bool;
      Condition_Enable_ULW : Bool;
      Condition_Enable_LLW : Bool;
      Condition_Enable_LLA : Bool;
   END_VAR


BEGIN
	(*
	Network 1: Start up
	*)
	IF #RESTART= true THEN
	  #QOUT:= 0;
	  #OPdwCmd:=0;
	END_IF;
	
	(*
	Network 2: Simulation On/Off
	Vaiable: OPdwCmd  Bit:  20  =  Process
	Vaiable: OPdwCmd  Bit:  21  =  Simulation
	*)
	IF (#LIOP_SEL=true AND #L_SIM=true) OR (#OPdwCmd.%X21=true AND #LIOP_SEL=false) THEN
	  #QSIM:=true;
	  #OPdwCmd.%X20:=false;
	  #OPdwCmd.%X21:=false;
	ELSIF (#LIOP_SEL=true AND #L_SIM=false) OR (#OPdwCmd.%X20=true AND #LIOP_SEL=false) THEN
	  #QSIM:= false;
	  #OPdwCmd.%X20:=false;
	  #OPdwCmd.%X21:=false;
	END_IF;
	
	(*
	Network 3: Mode limit Hysteresis
	Vaiable: OPdwCmd  Bit:  12  =  Hysteresis Percental
	Vaiable: OPdwCmd  Bit:  13  =  Hysteresis Absolute
	*)
	IF (#LIOP_SEL=true AND #LIM_HYS_Set=true) OR (#OPdwCmd.%X13=true AND #LIOP_SEL=false) THEN
	  #QLIM_HYS_Set:=true;
	  #OPdwCmd.%X12:=false;
	  #OPdwCmd.%X13:=false;
	ELSIF (#LIOP_SEL=true AND #LIM_HYS_Set=false) OR (#OPdwCmd.%X12=true AND #LIOP_SEL=false) THEN
	  #QLIM_HYS_Set:=false;
	  #OPdwCmd.%X12:=false;
	  #OPdwCmd.%X13:=false;
	END_IF;
	
	(*
	Network 4: Mode Periphery / Real value
	Vaiable: OPdwCmd  Bit:  14  =  Periphery
	Vaiable: OPdwCmd  Bit:  15  =  Real value
	*)
	IF (#LIOP_SEL=true AND #IN_MODE=true) OR (#OPdwCmd.%X15=true AND #LIOP_SEL=false) THEN
	  #QIN_MODE:=true;
	  #OPdwCmd.%X14:=false;
	  #OPdwCmd.%X15:=false;
	ELSIF (#LIOP_SEL=true AND #IN_MODE=false) OR (#OPdwCmd.%X14=true AND #LIOP_SEL=false) THEN
	  #QIN_MODE:=false;
	  #OPdwCmd.%X14:=false;
	  #OPdwCmd.%X15:=false;
	END_IF;
	
	(*
	Network 5: Reset Operation
	Vaiable: OPdwCmd  Bit:  24  =  Reset
	*)
	// Rising edge by linking
	IF #L_RESET=true AND #Condition_SEF_L_RESET_Link=false THEN
	  #SEF_L_RESET_Link:=true;
	  #Condition_SEF_L_RESET_Link:=true;
	ELSIF #L_RESET=true AND #Condition_SEF_L_RESET_Link=true THEN
	  #SEF_L_RESET_Link:=false;
	ELSE
	  #Condition_SEF_L_RESET_Link:=false;
	END_IF;
	// Rising edge by operator
	IF #OPdwCmd.%X24=true THEN
	  #SEF_L_RESET_OP:=true;
	  #OPdwCmd.%X24:=false;
	ELSE
	  #SEF_L_RESET_OP:=false;
	END_IF;
	// Reset error
	#OP_RESET:=(#LIOP_SEL=true AND #SEF_L_RESET_Link=true) OR (#SEF_L_RESET_OP=true AND #LIOP_SEL=false);
	
	(*
	Network 6: Enable alarm for upper limit
	Vaiable: OPdwCmd  Bit:  0  =  Enable alarm upper limit
	*)
	IF #OPdwCmd.%X0=true THEN
	  #Condition_Enable_ULA:=NOT #Condition_Enable_ULA;
	  #OPdwCmd.%X0:=false;
	END_IF;
	
	IF (#LIOP_SEL=true AND #LIM_ULA_Enable=true) OR (#LIOP_SEL=false AND #Condition_Enable_ULA=true) THEN  
	  #QLIM_ULA_Enable:=true;
	ELSIF (#LIOP_SEL=true AND #LIM_ULA_Enable=false) OR (#LIOP_SEL=false AND #Condition_Enable_ULA=false) THEN
	  #QLIM_ULA_Enable:=false;
	END_IF;
	
	  
	(*
	Network 7: Enable warning for upper limit
	Vaiable: OPdwCmd  Bit:  1  =  Enable warning upper limit
	*)
	IF #OPdwCmd.%X1=true THEN
	  #Condition_Enable_ULW:=NOT #Condition_Enable_ULW;
	  #OPdwCmd.%X1:=false;
	END_IF;
	
	IF (#LIOP_SEL=true AND #LIM_ULW_Enable=true) OR (#LIOP_SEL=false AND #Condition_Enable_ULW=true) THEN  
	  #QLIM_ULW_Enable:=true;
	ELSIF (#LIOP_SEL=true AND #LIM_ULW_Enable=false) OR (#LIOP_SEL=false AND #Condition_Enable_ULW=false) THEN
	  #QLIM_ULW_Enable:=false;
	END_IF;
	
	(*
	Network 8: Enable warning for lower limit
	Vaiable: OPdwCmd  Bit:  2  =  Enable warning lower limit
	*)
	IF #OPdwCmd.%X2=true THEN
	  #Condition_Enable_LLW:=NOT #Condition_Enable_LLW ;
	  #OPdwCmd.%X2:=false;
	END_IF;
	
	IF (#LIOP_SEL=true AND #LIM_LLW_Enable=true) OR (#LIOP_SEL=false AND #Condition_Enable_LLW=true) THEN  
	  #QLIM_LLW_Enable:=true;
	ELSIF (#LIOP_SEL=true AND #LIM_LLW_Enable=false) OR (#LIOP_SEL=false AND #Condition_Enable_LLW=false) THEN
	  #QLIM_LLW_Enable:=false;
	END_IF;
	
	(*
	Network 9: Enable alarm for lower limit
	Vaiable: OPdwCmd  Bit:  3  =  Enable alarm lower limit
	*)
	IF #OPdwCmd.%X3=true THEN
	  #Condition_Enable_LLA:=NOT #Condition_Enable_LLA;
	  #OPdwCmd.%X3:=false;
	END_IF;
	
	IF (#LIOP_SEL=true AND #LIM_LLA_Enable=true) OR (#LIOP_SEL=false AND #Condition_Enable_LLA=true) THEN  
	  #QLIM_LLA_Enable:=true;
	ELSIF (#LIOP_SEL=true AND #LIM_LLA_Enable=false) OR (#LIOP_SEL=false AND #Condition_Enable_LLA=false) THEN
	  #QLIM_LLA_Enable:=false;
	END_IF;
	
	(*
	Network 10: Calculate hysteresis value
	*)
	IF #LIOP_SEL=true AND #QLIM_HYS_Set=true THEN
	  // Absolute by PLC
	  #OP_HI_LIM:=#HI_LIM;
	  #OP_LO_LIM:=#LO_LIM;
	  #OP_LIM_HYS_Perc:=#LIM_HYS/((#HI_LIM-#LO_LIM)/100);
	  #OP_LIM_HYS_Abs:=#LIM_HYS;
	  #QHI_LIM:=#HI_LIM;
	  #QLO_LIM:=#LO_LIM;
	  #QLIM_HYS:=#OP_LIM_HYS_Abs;
	ELSIF #LIOP_SEL=true AND #QLIM_HYS_Set=false THEN
	  // Percental by PLC
	  #OP_HI_LIM:=#HI_LIM;
	  #OP_LO_LIM:=#LO_LIM;
	  #OP_LIM_HYS_Perc:=#LIM_HYS;
	  #OP_LIM_HYS_Abs:=#LIM_HYS*((#HI_LIM-#LO_LIM)/100);
	  #QHI_LIM:=#HI_LIM;
	  #QLO_LIM:=#LO_LIM;
	  #QLIM_HYS:=#OP_LIM_HYS_Abs;
	ELSIF #LIOP_SEL=false AND #QLIM_HYS_Set=true THEN
	  // Absolute by operator
	  #QHI_LIM:=#OP_HI_LIM;
	  #QLO_LIM:=#OP_LO_LIM;
	  #OP_LIM_HYS_Perc:=#OP_LIM_HYS_Abs/((#OP_HI_LIM-#OP_LO_LIM)/100);
	  #QLIM_HYS:=#OP_LIM_HYS_Abs;
	ELSE
	  // Percental by operator
	  #QHI_LIM:=#OP_HI_LIM;
	  #QLO_LIM:=#OP_LO_LIM;
	  #OP_LIM_HYS_Abs:=#OP_LIM_HYS_Perc*((#OP_HI_LIM-#OP_LO_LIM)/100);
	  #QLIM_HYS:=#OP_LIM_HYS_Abs;
	END_IF;
	
	//Transfer output to simulation value in process mode
	IF #QSIM=false THEN
	  #IN_SIM:=#QOUT;
	END_IF;
	(*
	Network 11: Convert integer to real and scale it to selcted mode
	*)
	IF #QIN_MODE=false AND #QSIM=false AND #BIPOLAR=false THEN
	  // Convert integer to real and scale in unipolar mode (4..20mA)
	  #QOUT:=(INT_TO_REAL(#IN_INT)/27648*(#HI_LIM-#LO_LIM))+#LO_LIM;
	ELSIF #QIN_MODE=false AND #QSIM=false AND #BIPOLAR=true THEN
	  // Convert integer to real and scale in bipolar mode (4..20mA)
	  #QOUT:=(((INT_TO_REAL(#IN_INT)+27648)/55296)*(#HI_LIM-#LO_LIM))+#LO_LIM;
	END_IF;
	
	//Che errors
	#QERR_EXT:=#ERR_EXTERN;
	#QLOCK:=#LOCK;
	
	(*
	Network 12: Check errors for simulation mode or real value
	*)
	IF (#QIN_MODE=true OR #QSIM=true) AND #QHI_LIM>=#QOUT AND #QLO_LIM<=#QOUT THEN
	    #QERR_OVERRUN:=false;
	    #QERR_HIGHRANGE:=false;
	    #QERR_LOWRANGE:=false;
	    #QERR_WIRE:=false;
	  END_IF;
	
	(*
	Network 13: Check errors for periphery unipolar mode (4..20mA)
	*)
	(*
	    Measuring Range   Units       Range
	    (4..20mA)         (Dez)
	    ============================================
	    >22,81            >32511      Overrun
	    --------------------------------------------
	    22,81              32511
	      .                           High range
	    20,01              27649         
	    --------------------------------------------
	    20,00              27648 
	      .                           Nominal range
	     4,00                  0
	    --------------------------------------------
	     3,99                 -1
	      .                           Low range
	     1,185             -4864
	    --------------------------------------------
	    <1,185            <-4864      Wire breakage
	*)
	IF #QSIM=false AND #QIN_MODE=false AND #BIPOLAR=false THEN
	  CASE #IN_INT OF
	    -4864..-1:      // Low range
	    #QERR_OVERRUN:=false;
	    #QERR_HIGHRANGE:=false;
	    #QERR_LOWRANGE:=true;
	    #QERR_WIRE:=false;
	    0..27648:       // Nominal range
	    #QERR_OVERRUN:=false;
	    #QERR_HIGHRANGE:=false;
	    #QERR_LOWRANGE:=false;
	    #QERR_WIRE:=false;
	    27649..32511:   // High range
	    #QERR_OVERRUN:=false;
	    #QERR_HIGHRANGE:=true;
	    #QERR_LOWRANGE:=false;
	    #QERR_WIRE:=false;
	  ELSE
	    IF #IN_INT>32511 THEN
	      // Overrun
	      #QERR_OVERRUN:=true;
	      #QERR_HIGHRANGE:=false;
	      #QERR_LOWRANGE:=false;
	      #QERR_WIRE:=false;
	    ELSE
	      // Wire breakage
	      #QERR_OVERRUN:=false;
	      #QERR_HIGHRANGE:=false;
	      #QERR_LOWRANGE:=false;
	      #QERR_WIRE:=true;
	    END_IF;  
	  END_CASE;
	END_IF;
	
	(*
	Network 14: Check errors for periphery bipolar mode (4..20mA)
	*)
	(*
	    Measuring Range   Units       Range
	    (4..20mA)         (Dez)
	    ============================================
	    >22,81            >32511      Overrun
	    --------------------------------------------
	    22,81              32511
	      .                           High range
	    20,01              27649         
	    --------------------------------------------
	    20,00              27648 
	      .                           Nominal range
	     4,00             -27648
	    --------------------------------------------
	     3,99             -27649
	      .                           Low range
	     1,185            -32512
	    --------------------------------------------
	    <1,185           <-32512      Wire breakage
	*)
	IF #QSIM=false AND #QIN_MODE=false AND #BIPOLAR=true THEN
	  CASE #IN_INT OF
	    -32512..-27649:         // Low range
	    #QERR_OVERRUN:=false;
	    #QERR_HIGHRANGE:=false;
	    #QERR_LOWRANGE:=true;
	    #QERR_WIRE:=false;
	    -27648..27648:         // Nominal range
	    #QERR_OVERRUN:=false;
	    #QERR_HIGHRANGE:=false;
	    #QERR_LOWRANGE:=false;
	    #QERR_WIRE:=false;
	    27649..32511:         // High range
	    #QERR_OVERRUN:=false;
	    #QERR_HIGHRANGE:=true;
	    #QERR_LOWRANGE:=false;
	    #QERR_WIRE:=false;
	  ELSE
	    IF #IN_INT>32511 THEN
	      // Overrun
	      #QERR_OVERRUN:=true;
	      #QERR_HIGHRANGE:=false;
	      #QERR_LOWRANGE:=false;
	      #QERR_WIRE:=false;
	    ELSE
	      // Wire breakage
	      #QERR_OVERRUN:=false;
	      #QERR_HIGHRANGE:=false;
	      #QERR_LOWRANGE:=false;
	      #QERR_WIRE:=true;
	    END_IF;  
	  END_CASE;
	END_IF;
	
	(*
	Network 15: Check range error for real value
	*)
	//  Check for high range injury
	IF (#IN>#QHI_LIM AND #QIN_MODE=true AND #QSIM=false AND #LIOP_SEL=true) OR
	   (#IN_SIM>#QHI_LIM AND #QSIM=true AND #LIOP_SEL=true) OR
	   (#OP_SIM_Value>#QHI_LIM AND #QSIM=true AND #LIOP_SEL=false) THEN
	      #QERR_HIGHRANGE:=true;
	END_IF;
	//  Check for low range injury
	IF (#IN<#QLO_LIM AND #QIN_MODE=true AND #QSIM=false AND #LIOP_SEL=true) OR
	   (#IN_SIM<#QLO_LIM AND #QSIM=true AND #LIOP_SEL=true) OR
	   (#OP_SIM_Value<#QLO_LIM AND #QSIM=true AND #LIOP_SEL=false) THEN
	      #QERR_LOWRANGE:=true;
	END_IF;
	    
	(*
	Network 16: General Error
	*)
	IF #OP_RESET=true THEN
	  #QERR:=false;
	ELSIF #QERR_EXT=true OR #QLOCK=true OR #QERR_OVERRUN OR #QERR_WIRE THEN
	  #QERR:=true;
	END_IF;
	
	(*
	Network 17: Upper limit alarm
	*)
	IF #QLIM_ULA_Enable=true THEN
	  IF #QLIM_ULA<=#QOUT THEN
	    #QALARM_UL:=true;
	  ELSIF (#QLIM_ULA-#QLIM_HYS)>#QOUT THEN
	    #QALARM_UL:=false;
	  END_IF;
	ELSE
	  #QALARM_UL:=false;
	END_IF;
	 
	(*
	Network 18: Upper limit warning
	*)
	IF #QLIM_ULW_Enable=true THEN
	  IF #QLIM_ULW<=#QOUT THEN
	    #QWARN_UL:=true;
	  ELSIF (#QLIM_ULW-#QLIM_HYS)>#QOUT THEN
	    #QWARN_UL:=false;
	  END_IF;
	ELSE
	  #QWARN_UL:=false;
	END_IF;
	
	(*
	Network 19: Lower limit warning
	*)
	IF #QLIM_LLW_Enable=true THEN
	  IF #QLIM_LLW>=#QOUT THEN
	    #QWARN_LL:=true;
	  ELSIF (#QLIM_LLW+#QLIM_HYS)<#QOUT THEN
	    #QWARN_LL:=false;
	  END_IF;
	ELSE
	  #QWARN_LL:=false;
	END_IF;
	
	(*
	Network 20: Lower limit alarm
	*)
	IF #QLIM_LLA_Enable=true THEN
	  IF #QLIM_LLA>=#QOUT THEN
	    #QALARM_LL:=true;
	  ELSIF (#QLIM_LLA+#QLIM_HYS)<#QOUT THEN
	    #QALARM_LL:=false;
	  END_IF;
	ELSE
	  #QALARM_LL:=false;
	END_IF;
	
	(*
	Network 21: Set limit value
	*)
	IF #QSIM=true AND #LIOP_SEL=false THEN
	  // Set values in simulation mode by operator
	  #QHI_LIM:=#OP_HI_LIM;
	  #QLO_LIM:=#OP_LO_LIM;
	  #QLIM_ULA:=#OP_LIM_ULA;
	  #QLIM_ULW:=#OP_LIM_ULW;
	  #QLIM_LLW:=#OP_LIM_LLW;
	  #QLIM_LLA:=#OP_LIM_LLA;
	ELSE
	  // Set values in normal mode by linking
	  #OP_HI_LIM:=#HI_LIM;
	  #QHI_LIM:=#HI_LIM;
	  #OP_LO_LIM:=#LO_LIM;
	  #QLO_LIM:=#LO_LIM;
	  #OP_LIM_ULA:=#LIM_ULA;
	  #QLIM_ULA:=#LIM_ULA;
	  #OP_LIM_ULW:=#LIM_ULW;
	  #QLIM_ULW:=#LIM_ULW;
	  #OP_LIM_LLW:=#LIM_LLW;
	  #QLIM_LLW:=#LIM_LLW;
	  #OP_LIM_LLA:=#LIM_LLA;
	  #QLIM_LLA:=#LIM_LLA;
	END_IF;
	
	(*
	Network 22: Check settings and values
	*)
	IF #QSIM=false AND #QIN_MODE=true THEN
	  // Set settings in process mode by PLC (real value)
	  #QOUT:=#IN;
	ELSIF #QSIM=true AND #LIOP_SEL=false THEN
	  // Set settings in simulation mode by operator (real value)
	  #QOUT:=#OP_SIM_Value;
	ELSIF #QSIM=true AND #LIOP_SEL=true THEN
	  // Set settings in simulation mode by PLC (real value)
	  #QOUT:=#IN_SIM;
	END_IF;
	
	IF #QSIM=false AND #LIOP_SEL=true AND #IN_MODE=false THEN
	  //Set settings in process mode by PLC (periphery)
	  IF #QERR_EXT=true OR #QLOCK=true THEN
	  //Set value in case of error
	    #QOUT:=#QLO_LIM;
	ELSE
	  IF #QOUT>#QHI_LIM THEN
	    #QOUT:=#QHI_LIM;
	  ELSIF #QOUT<#LO_LIM THEN
	    #QOUT:=#QLO_LIM;
	  END_IF;
	END_IF;
	END_IF;
	(*
	Network 23: Infuence visibility of faceplate window
	*)
	IF #OP_VISIBILITY<>#VISIBILITY_OLD THEN
	  #VISIBILITY_OLD:=#OP_VISIBILITY;
	  #VISIBILITY:=#OP_VISIBILITY;
	ELSIF #VISIBILITY<>#VISIBILITY_OLD THEN
	  #VISIBILITY_OLD:=#VISIBILITY;
	  #OP_VISIBILITY:=#VISIBILITY;
	END_IF;
	
	(*
	Network 24: Transfer output to simulation value in process mode
	*)
	IF #QSIM=false THEN
	  #IN_SIM:=#QOUT;
	END_IF;
	
	(*
	Network 25: Check errors
	*)
	#QERR_EXT:=#ERR_EXTERN;
	#QLOCK:=#LOCK;
	
	(*
	Network 26: Set state for HMI
	*)
	#QdwState.%X0:= #QIN_MODE;
	#QdwState.%X1:=#QLIM_HYS_Set;
	#QdwState.%X2:=false;
	#QdwState.%X3:=false;
	#QdwState.%X4:=#QLIM_ULA_Enable;
	#QdwState.%X5:=#QLIM_ULW_Enable;
	#QdwState.%X6:=#QLIM_LLW_Enable;
	#QdwState.%X7:=#QLIM_LLA_Enable;
	#QdwState.%X9:=#QALARM_LL OR #QALARM_UL;
	#QdwState.%X8:=NOT #QdwState.%X9 AND (#QWARN_LL OR #QWARN_UL);
	#QdwState.%X10:=false;
	#QdwState.%X11:=false;
	#QdwState.%X12:=#QERR_LOWRANGE;
	#QdwState.%X13:=#QERR_HIGHRANGE;
	#QdwState.%X14:=#QERR_OVERRUN;
	#QdwState.%X15:=#QERR_WIRE;
	#QdwState.%X16:=false;
	#QdwState.%X17:=false;
	#QdwState.%X18:=#QSIM;
	#QdwState.%X19:=false;
	#QdwState.%X20:=false;
	#QdwState.%X21:=false;
	#QdwState.%X22:=false;
	#QdwState.%X23:=false;
	#QdwState.%X24:=#QERR;
	#QdwState.%X25:=#QERR_EXT;
	#QdwState.%X26:=#QLOCK;
	#QdwState.%X27:=#LOCK;
	#QdwState.%X28:=false;
	#QdwState.%X29:=false;
	#QdwState.%X30:=false;
	#QdwState.%X31:=false;
	
	(*
	Network 27: Bit alarm procedure
	*)
	#QwAlarm.%X0:=#QALARM_LL;
	#QwAlarm.%X1:=#QALARM_UL;
	#QwAlarm.%X2:=false;
	#QwAlarm.%X3:=false;
	#QwAlarm.%X4:=#QLOCK;
	#QwAlarm.%X5:=false;
	#QwAlarm.%X6:=#QERR_EXT;
	#QwAlarm.%X7:=#QERR;
	#QwAlarm.%X8:=#QWARN_LL;
	#QwAlarm.%X9:=#QWARN_UL;
	#QwAlarm.%X10:=false;
	#QwAlarm.%X11:=false;
	#QwAlarm.%X12:=#LOCK;
	#QwAlarm.%X13:=false;
	#QwAlarm.%X14:=false;
	#QwAlarm.%X15:=#QSIM;
	
END_FUNCTION_BLOCK

FUNCTION_BLOCK "Digital_1"
TITLE =  Digital
{ S7_Optimized_Access := 'FALSE' }
AUTHOR : RM
FAMILY : MON
VERSION : 0.1
//Interface for a binary value  
   VAR_INPUT 
      LOCK : Bool;   // 1 = Inerlock active
      ERR_EXTERN : Bool;   // 1 = External error arised
      LIOP_SEL : Bool;   // 0 = Operator; 1 = Linking
      L_SIM : Bool;   // 0 = Normal; 1 = Simulation
      L_RESET : Bool;   // 1 = Reset error peripherie
      INP : Bool;   // 1 = Digital input signal is ON
      INP_NEG : Bool;   // 1 = Negation input signal is ACTIVE
      INP_SIM : Bool;   // 1 = Digital simulation signal is ON
      DELAY_TIME : Time := T#5S;   // Delay time of setting bit
      DELAY_TIME_OFF : Time := T#5S;   // Delay time of resetting bit
      INSTANCE : String[254] := 'Digital_001';   // Filter attribute for message view, also used for labelling
      RESTART : Bool;   // 1 = Initialize FB at startup (first cycle fo PLC)
   END_VAR

   VAR_OUTPUT 
      QdwState : DWord;   // Status HMI
      QLOCK : Bool;   // 1 = Interlock is active
      QSIM : Bool;   // 0 = Normal; 1 = Simulation
      QON : Bool;   // 1 = On
      QON_DELAY : Bool;   // 1 = On with delay
      QOFF : Bool;   // 1 = Off
      QOFF_DELAY : Bool;   // 1 = Off with delay
      QOUT : Bool;   // 1 = On or 1 = Off with delay, DI Out with Time Delay
      QDELAY_TIME : Time;   // Delay time for switching ON
      QDELAY_TIME_OFF : Time;   // Delay time for switching OFF
      QINP : Bool;   // 1 = Input signal including negation information
      QERR : Bool;   // 1 = Common error
      QERR_EXTERN : Bool;   // 1 = External error
      QwAlarm : Word;   // Bit alarm producere
   END_VAR

   VAR_IN_OUT 
      VISIBILITY : Byte;   // Bit 0: Tab1 of window; Bit 1: Tab2 of window; ... ; Bit 7: Minimize
      OPdwCmd : DWord;   // Control word from HMI
   END_VAR

   VAR 
      OP_RESET : Bool;   // Reset error
      OP_VISIBILITY : Byte;   // Operator: Bit 0: Tab1 of window; Bit 1: Tab2 of window; ... ; Bit 7: Minimize
      VISIBILITY_OLD : Byte;   // Save last status of VISIBILITY
      DELAY_ON : Bool;   // Delay for switching ON required
      DELAY_OFF : Bool;   // Delay for switching OFF required
      SE_L_RESET_LINK : Bool;   // Signal edge for the reset input from linking
      SE_L_RESET_LINK_COND : Bool;   // Condition of signal edge
      SE_L_RESET_OP : Bool;   // Signal edge for the reset input from operator
      T_ON {InstructionName := 'TON_TIME'; LibVersion := '1.0'} : TON_TIME;
      T_OFF {InstructionName := 'TON_TIME'; LibVersion := '1.0'} : TON_TIME;   // Timer instance for turning off
      OLD_SIG_COND : Bool;   // Condition of the old signal
      SINP_SIM : Bool;   // Signal from operator in simulation mode
   END_VAR

   VAR_TEMP 
      TIMER_ON : Bool;   // Timer signal ON
      TIMER_OFF : Bool;   // Timer signal OFF
   END_VAR


BEGIN
	
	(*
	Network 1: Start up
	*)
	IF #RESTART= true THEN
	  #QON:= false;
	  #QON_DELAY:=false;
	  #QOFF:=true;
	  #QOFF_DELAY:=false;
	  #OPdwCmd:=0;
	END_IF;
	
	(*
	Network 2: Simulation On/Off
	Vaiable: OPdwCmd  Bit:  20  =  Process
	Vaiable: OPdwCmd  Bit:  21  =  Simulation
	*)
	IF (#LIOP_SEL=true AND #L_SIM=true) OR (#OPdwCmd.%X21=true AND #LIOP_SEL=false) THEN
	  #QSIM:=true;
	  #OPdwCmd.%X20:=false;
	  #OPdwCmd.%X21:=false;
	ELSIF (#LIOP_SEL=true AND #L_SIM=false) OR (#OPdwCmd.%X20=true AND #LIOP_SEL=false) THEN
	  #QSIM:= false;
	  #OPdwCmd.%X20:=false;
	  #OPdwCmd.%X21:=false;
	END_IF;
	
	(*
	Network 3: Reset Operation
	Vaiable: OPdwCmd  Bit:  24  =  Reset
	*)
	// Rising edge by linking
	IF #L_RESET=true AND #SE_L_RESET_LINK_COND=false THEN
	  #SE_L_RESET_LINK:=true;
	  #SE_L_RESET_LINK_COND:=true;
	ELSIF #L_RESET=true AND #SE_L_RESET_LINK_COND=true THEN
	  #SE_L_RESET_LINK:=false;
	ELSE
	  #SE_L_RESET_LINK_COND:=false;
	END_IF;
	// Rising edge by operator
	IF #OPdwCmd.%X24=true THEN
	  #SE_L_RESET_OP:=true;
	  #OPdwCmd.%X24:=false;
	ELSE
	  #SE_L_RESET_OP:=false;
	END_IF;
	// Reset error
	#OP_RESET:=(#SE_L_RESET_LINK=TRUE) OR (#SE_L_RESET_OP AND NOT #LIOP_SEL);
	
	(*
	Network 4: Create input signal
	*)
	#QINP:=#INP XOR #INP_NEG;
	
	(*
	Network 6: Check errors
	*)
	#QERR_EXTERN:=#ERR_EXTERN;
	// Check for interlock
	IF #LOCK=true AND (#QON=true OR #QON_DELAY=true OR #QOFF_DELAY=true) THEN
	  #QLOCK:=true;
	ELSIF #OP_RESET=true THEN
	  #QLOCK:=false;
	END_IF;
	// Check for general error
	IF #QERR_EXTERN=true OR #QLOCK=true THEN
	  #QERR:=true;
	ELSIF #OP_RESET=true THEN
	  #QERR:=false;
	END_IF;
	
	(*
	Network 7: TOGGLE Simulation Bit
	*)
	IF #OPdwCmd.%X4=true AND #QSIM=true THEN
	  #SINP_SIM := NOT #SINP_SIM;
	  #OPdwCmd.%X4:=false;
	END_IF;
	
	(*
	Network 8: Bumpless switch to simulation mode
	*)
	IF #QSIM=false THEN
	    #INP_SIM := #QINP;  
	END_IF;
	
	(*
	Network 9: Evaluate for delays
	*)
	// Evaluate for ON delay
	IF #DELAY_TIME<> t#1ms THEN
	  #DELAY_ON:=true;
	ELSE
	  #DELAY_ON:=false; 
	END_IF;
	// Evaluate for OFF delay
	IF #DELAY_TIME_OFF <> t#1ms THEN
	  #DELAY_OFF:=true;
	ELSE
	  #DELAY_OFF:=false;
	END_IF;
	
	(*
	Network 10: Settting ON/OFF
	*)
	// Delay time for setting on
	    #T_ON(IN:=#DELAY_ON AND #QON_DELAY,
	           PT:=#DELAY_TIME,
	           Q=>#TIMER_ON,
	           ET=>#QDELAY_TIME);
	// Delay time for setting off               
	    #T_OFF(IN:=#DELAY_OFF AND #QOFF_DELAY ,
	            PT:=#DELAY_TIME_OFF,
	            Q=>#TIMER_OFF,
	            ET=>#QDELAY_TIME_OFF);
	
	IF #QERR=false AND #LOCK=false THEN
	  // Sets variable, for closing process in progress
	  #QON_DELAY:=((NOT #QSIM AND #QINP) OR (#QSIM AND (#INP_SIM OR #SINP_SIM)))AND NOT #QON;
	  // Sets variable, for opening process in progress
	  #QOFF_DELAY:=((NOT #QSIM AND NOT #QINP) OR (#QSIM AND NOT (#INP_SIM OR #SINP_SIM)))AND NOT #QOFF;
	
	  // Sets variable, for ON/OFF   
	  IF #TIMER_ON=true OR (#QINP=true AND #DELAY_ON=false) OR (#OLD_SIG_COND=true AND #QOFF_DELAY=false) THEN
	    // On case
	     #QON:=true;
	     #QOFF:=false;
	     #OLD_SIG_COND:=true;
	   ELSIF #TIMER_OFF=true OR (#QINP=false AND #DELAY_OFF=false) OR (#OLD_SIG_COND=false AND #QON_DELAY=false) THEN
	     // Off case
	     #QON:=false;
	     #QOFF:=true;
	     #OLD_SIG_COND:=false;
	   ELSE
	     // switch ON <--> OFF case
	     #QON:=false;
	     #QOFF:=false;
	   END_IF;
	ELSE
	   // Error case
	     #QON_DELAY:=false;
	     #QOFF_DELAY:=false;
	     #QON:=false;
	     #QOFF:=NOT #QERR;
	     #OLD_SIG_COND:=false;
	END_IF;
	
	(*
	Network 11: QOUT
	*)
	#QOUT := #QON OR #QOFF_DELAY;
	
	(*
	Network 12: Influence visibility of faceplate window
	*)
	IF #OP_VISIBILITY<>#VISIBILITY_OLD THEN
	  #VISIBILITY_OLD:=#OP_VISIBILITY;
	  #VISIBILITY:=#OP_VISIBILITY;
	ELSIF #VISIBILITY<>#VISIBILITY_OLD THEN
	  #VISIBILITY_OLD:=#VISIBILITY;
	  #OP_VISIBILITY:=#VISIBILITY;
	END_IF;
	
	(*
	Network 13: Set state for HMI
	*)
	#QdwState.%X0:=#QOFF;
	#QdwState.%X1:=#QOFF_DELAY;
	#QdwState.%X2:=#QON;
	#QdwState.%X3:=#QON_DELAY;
	#QdwState.%X4:=false;
	#QdwState.%X5:=false;
	#QdwState.%X6:=false;
	#QdwState.%X7:=false;
	#QdwState.%X8:=#QINP;
	#QdwState.%X9:=false;
	#QdwState.%X10:=false;
	#QdwState.%X11:=false;
	#QdwState.%X12:=#INP_NEG;
	#QdwState.%X13:=#SINP_SIM;
	#QdwState.%X14:=false;
	#QdwState.%X15:=false;
	#QdwState.%X16:=false;
	#QdwState.%X17:=false;
	#QdwState.%X18:=#QSIM;
	#QdwState.%X19:=false;
	#QdwState.%X20:=false;
	#QdwState.%X21:=false;
	#QdwState.%X22:=false;
	#QdwState.%X23:=false;
	#QdwState.%X24:=#QERR;
	#QdwState.%X25:=#QERR_EXTERN;
	#QdwState.%X26:=#QLOCK;
	#QdwState.%X27:=#LOCK;
	#QdwState.%X28:=false;
	#QdwState.%X29:=false;
	#QdwState.%X30:=false;
	#QdwState.%X31:=false;
	
	(*
	Network 14: Bit alarm procedure
	*)
	#QwAlarm.%X0:=false;
	#QwAlarm.%X1:=false;
	#QwAlarm.%X2:=false;
	#QwAlarm.%X3:=false;
	#QwAlarm.%X4:=#QLOCK;
	#QwAlarm.%X5:=false;
	#QwAlarm.%X6:=#QERR_EXTERN;
	#QwAlarm.%X7:=#QERR;
	#QwAlarm.%X8:=#QON;
	#QwAlarm.%X9:=#QON_DELAY;
	#QwAlarm.%X10:=false;
	#QwAlarm.%X11:=false;
	#QwAlarm.%X12:=#LOCK;
	#QwAlarm.%X13:=false;
	#QwAlarm.%X14:=false;
	#QwAlarm.%X15:=#QSIM;
END_FUNCTION_BLOCK

FUNCTION_BLOCK "Motor_w_VSD_Sinamics"
TITLE = Motor
{ S7_Optimized_Access := 'FALSE' }
AUTHOR : RM
VERSION : 0.1
//Interface FB for a motor
   VAR_INPUT 
      LOCK : Bool;   // 1 = Interlock active
      ERR_EXTERN : Bool;   // 1 = External error arised
      LIOP_SEL : Bool;   // 0 = Operator; 1 = Linking
      L_AUT : Bool;   // 0 = Manual; 1 = Automatic
      L_REMOTE : Bool;   // 0 = Local; 1 = Remote
      L_SIM : Bool;   // 0 = Normal; 1 = Simulation
      L_RESET : Bool;   // 1 = Reset error peripherie
      AUT_ON : Bool;   // 1 = CMD ON Automatic
      MAN_ON : Bool;   // 1 = CMD ON Manual
      SIM_ON : Bool;   // 1 = CMD ON Simulation
      FB_MODE : Bool;   // 0 = FB Run from communication ,1 = FB_ON
      FB_ON : Bool;   // 1 = Feedback Motor ON
      drive_reversing : Bool;
      L_MON : Bool;   // 1 = Monitoring ON
      MON_T : Time := t#5s;   // Monitoring starting time in process mode
      MON_T_STOP : Time := t#5s;   // Monitoring stopping time in process mode
      MPS : Bool;   // 1 = Motor protection switch ON
      L_FLOW_MON : Bool;   // 1 = Monitoring flow
      FLOW : Real;   // Current flow
      FLOW_LL : Real := 5.0;   // Low level flow
      FLOW_MT : Time := t#8s;   // Delay of monitoring lower flow
      IN_SP_Speed : Real;   // Setpoint Speed in Percen
      IN_SW : Word;   // IN Status word from Drive
      "IN _AV" : Int;   // IN Actual Speed from Drive
      IN_Volt : Int;   // IN Actual Voltage
      IN_Ampere : Int;   // IN Actual Ampere
      IN_KW : Int;   // IN Actual KW
      IN_Nm : Int;   // IN Actual Torque
      INSTANCE : String := 'Motor_001';   // Filter attribute for message view, also used for labelling
      RESTART : Bool;   // 1 = Initialize FB at startup (first cycle of PLC)
   END_VAR

   VAR_OUTPUT 
      QdwState : DWord;   // Status HMI
      QwState : Int;   // Motor: 0 = Stop; 1 = Starting; 2 = Run; 3 = Stopping
      QSTOPPING : Bool;   // 1 = Stopping
      QSTOP : Bool;   // 1 = Stop
      QSTARTING : Bool;   // 1 = Starting
      QRUN : Bool;   // 1 = Run
      QCMD_ON : Bool;   // 0 = Stop; 1 = Start (automatic & manual mode)
      QMON : Bool;   // 1 = Monitoring is ON
      QMON_ERR : Bool;   // 1 = Monitoring errror
      QMON_T : Time;   // Expierd starting time in process mode
      QMON_T_STOP : Time;   // Expierd stopping time in process mode
      QFLOW_MON : Bool;   // 1 = Flow monitoring is ON
      QFLOW_MT : Time;   // Expiered delay of monitoring lower flow
      QFLOW_ERR : Bool;   // 1 = Error flow monitoring
      QMPS : Bool;   // 1 = Motor protecting switch
      QMAN_AUT : Bool;   // 0 = Manual; 1 = Automatic
      QREMOTE : Bool;   // 0 = Local; 1 = Remote
      QSIM : Bool;   // 0 = Normal; 1 = Simulation
      QLOCK : Bool;   // 1 = Interlock is active
      QERR : Bool;   // 1 = Common error
      QERR_EXT : Bool;   // 1 = External error
      QDrive_Fault : Bool;
      QDrive_Alarm : Bool;
      QwAlarm : Word;   // Bit alarm procedure
      Q_CW : Word;   // Out Control Word for VSD
      Q_SP_Speed : Word;   // Out SP Speed for VSD
      QAct_Speed : Real;   // Drive Actual Speed
      QAct_Volt : Real;   // Drive Actual Voltage
      QAct_Amp : Real;   // Drive Actual Ampere
      QAct_KW : Real;   // Drive Actual KW
      QAct_Nm : Real;   // Drive Actual Torque
   END_VAR

   VAR_IN_OUT 
      VISIBILITY : Byte;   // Bit 0: Tab1 of window; Bit 1: Tab2 of window; ... ; Bit 7: Minimize
      OPdwCmd : DWord;   // Contorl word HMI
   END_VAR

   VAR 
      FB_SIM : Bool;
      SP_SpeedHz : Real;   // setengah dari 100%
      Drive_Actual_Speed : Real;   // Drive Actual Speed in Percen
      Drive_CW : Word;
      Drive_SW : Word;
      SIM_T : Time;
      QSIM_T : Time;
      SIM_T_STOP : Time;
      QSIM_T_STOP : Time;
      QCMD_SIM : Bool;
      OP_RESET : Bool;   // Reset errors
      QFLOW_MON_ACK : Bool;
      OP_VISIBILITY : Byte;   // Bit 0: Tab1 of window; Bit 1: Tab2 of window; ... ; Bit 7: Minimize
      VISIBILITY_OLD : Byte;   // Save last status of VISIBILITY
      QFB_RUN : Bool;
      Drive_FB_ON : Bool;   // Drive_Running
      Drive_Fault : Bool;   // Drive_Fault Active
      Drive_Alarm : Bool;   // Drive_Alarm Active
      SE_L_RESET_LINK : Bool;   // Signal edge for the reset input from linking
      SE_L_RESET_LINK_COND : Bool;   // Condition of signal edge
      SE_L_RESET_OP : Bool;   // Signal edge for the reset input from operator
      TSTARTING {InstructionName := 'TON_TIME'; LibVersion := '1.0'} : TON_TIME;
      TSTOPPING {InstructionName := 'TON_TIME'; LibVersion := '1.0'} : TON_TIME;
      TFLOW {InstructionName := 'TON_TIME'; LibVersion := '1.0'} : TON_TIME;
      TSTARTING_SIM {InstructionName := 'TON_TIME'; LibVersion := '1.0'} : TON_TIME;
      TSTOPPING_SIM {InstructionName := 'TON_TIME'; LibVersion := '1.0'} : TON_TIME;
   END_VAR

   VAR_TEMP 
      CON_ERR : Bool;   // Error in motor condition
      MON_ERR_STARTING : Bool;   // Monitoring error for starting motor in process mode
      MON_ERR_STOPPING : Bool;   // Monitoring error for stopping motor in process mode
      MON_SIM_STARTING : Bool;   // Monitoring error for starting motor in simulation mode
      MON_SIM_STOPPING : Bool;   // Monitoring error for stopping motor in simulation mode
      FB_ERR : Bool;   // Feedback error in process mode
      MON_ERR_FLOW2 : Bool;
      START_FLOW_TIME2 : Bool;
      START_FLOW_TIME : Bool;   // Start Signal of delay time for flow
      MON_ERR_FLOW : Bool;   // Monitoring error for flow
   END_VAR


BEGIN
	(********************************
	           Start up
	*********************************)
	IF #RESTART= true THEN
	  // Restart case
	  #QCMD_ON:= false;
	  #QSTOP:=true;
	  #QSTOPPING:=false;
	  #QRUN:=false;
	  #QSTARTING:=false;
	  #VISIBILITY:=0;
	  #OPdwCmd:=0;
	ELSE
	  // Normal case
	  
	  (******************************************
	    Network 1: Operating mode: manual/automatic
	    Vaiable: OPdwCmd  Bit:  16  =  Manual
	    Vaiable: OPdwCmd  Bit:  17  =  Automatic
	  *******************************************)
	  IF (#LIOP_SEL=true AND #L_AUT=true) OR (#OPdwCmd.%X17=true AND #LIOP_SEL=false) THEN
	    #QMAN_AUT:=true;
	    #OPdwCmd.%X16:=false;
	    #OPdwCmd.%X17:=false;
	  ELSIF (#LIOP_SEL=true AND #L_AUT=false) OR (#OPdwCmd.%X16=true AND #LIOP_SEL=false) THEN
	    #QMAN_AUT:= false;
	    #OPdwCmd.%X16:=false;
	    #OPdwCmd.%X17:=false;
	  END_IF;
	  
	  (******************************************
	    Network 2: Control mode: local/remote
	    Vaiable: OPdwCmd  Bit:  18  =  Local
	    Vaiable: OPdwCmd  Bit:  19  =  Remote
	  *******************************************)
	  IF (#LIOP_SEL=true AND #L_REMOTE=true) OR (#OPdwCmd.%X19=true AND #LIOP_SEL=false) THEN
	    #QREMOTE:=true;
	    #OPdwCmd.%X18:=false;
	    #OPdwCmd.%X19:=false;
	  ELSIF (#LIOP_SEL=true AND #L_REMOTE=false) OR (#OPdwCmd.%X18=true AND #LIOP_SEL=false) THEN
	    #QREMOTE:= false;
	    #OPdwCmd.%X18:=false;
	    #OPdwCmd.%X19:=false;
	  END_IF;
	  
	  (******************************************
	    Network 3: Simulation On/Off
	    Vaiable: OPdwCmd  Bit:  20  =  Process
	    Vaiable: OPdwCmd  Bit:  21  =  Simulation
	  *******************************************)
	  IF (#LIOP_SEL=true AND #L_SIM=true) OR (#OPdwCmd.%X21=true AND #LIOP_SEL=false) THEN
	    #QSIM:=true;
	    #OPdwCmd.%X20:=false;
	    #OPdwCmd.%X21:=false;
	  ELSIF (#LIOP_SEL=true AND #L_SIM=false) OR (#OPdwCmd.%X20=true AND #LIOP_SEL=false) THEN
	    #QSIM:= false;
	    #OPdwCmd.%X20:=false;
	    #OPdwCmd.%X21:=false;
	  END_IF;
	  
	  (*************************************
	    Network 4: Reset Operation
	    Vaiable: OPdwCmd  Bit:  24  =  Reset
	  **************************************)
	  // Rising edge by linking
	  IF #L_RESET=true AND #SE_L_RESET_LINK_COND=false THEN
	    #SE_L_RESET_LINK:=true;
	    #SE_L_RESET_LINK_COND:=true;
	  ELSIF #L_RESET=true AND #SE_L_RESET_LINK_COND=true THEN
	    #SE_L_RESET_LINK:=false;
	  ELSE
	    #SE_L_RESET_LINK_COND:=false;
	  END_IF;
	  // Rising edge by operator
	  IF #OPdwCmd.%X24=true THEN
	    #SE_L_RESET_OP:=true;
	    #OPdwCmd.%X24:=false;
	  ELSE
	    #SE_L_RESET_OP:=false;
	  END_IF;
	  // Reset error #OP_RESET:=((#LIOP_SEL AND #SE_L_RESET_LINK) OR (#SE_L_RESET_OP AND NOT #LIOP_SEL)) AND NOT #LOCK;
	  #OP_RESET:=(#SE_L_RESET_LINK=true) OR (#SE_L_RESET_OP AND NOT #LIOP_SEL) AND NOT #LOCK;
	  
	  (**********************************************
	    Network 5: Monitoring feedback ON/OFF
	    Vaiable: OPdwCmd  Bit:  8  =  Monitoring ON
	    Vaiable: OPdwCmd  Bit:  9  =  Monitoring OFF
	  ***********************************************)
	  IF (#LIOP_SEL=true AND #L_MON=false) OR (#OPdwCmd.%X9=true AND #LIOP_SEL=false)THEN
	    #QMON:=false;
	    #OPdwCmd.%X8:=false;
	    #OPdwCmd.%X9:=false;
	  ELSIF (#LIOP_SEL=true AND #L_MON=true) OR (#OPdwCmd.%X8=true AND #LIOP_SEL=false)THEN
	    #QMON:=true;
	    #OPdwCmd.%X8:=false;
	    #OPdwCmd.%X9:=false;
	  END_IF;
	  
	  (***************************************************
	    Network 6: Monitoring flow ON/OFF
	    Vaiable: OPdwCmd  Bit:  10  =  Monitoring flow ON
	    Vaiable: OPdwCmd  Bit:  11  =  Monitoring flow OFF
	  ****************************************************)
	  IF (#LIOP_SEL=true AND #L_FLOW_MON=false) OR (#OPdwCmd.%X11=true AND #LIOP_SEL=false)THEN
	    #QFLOW_MON:=false;
	    #OPdwCmd.%X10:=false;
	    #OPdwCmd.%X11:=false;
	  ELSIF (#LIOP_SEL=true AND #L_FLOW_MON=true) OR (#OPdwCmd.%X10=true AND #LIOP_SEL=false)THEN
	    #QFLOW_MON:=true;
	    #OPdwCmd.%X10:=false;
	    #OPdwCmd.%X11:=false;
	  END_IF;
	  
	   (**********************************************
	    Network 6: START/STOP Motor
	    Vaiable: OPdwCmd  Bit:  0  =  STOP Motor
	    Vaiable: OPdwCmd  Bit:  1  =  START Motor
	  ***********************************************)
	  IF #QERR=false THEN
	    // No errors occurs
	    IF #QSIM=false THEN
	     // Simulation mode is not active
	      // Automatic/Manual mode
	      IF #QMAN_AUT=true THEN
	        // Automatic mode is active
	        // OPEN/CLOSE valve by linking (AUT_ON)
	        #QCMD_ON:=#AUT_ON;
	        #OPdwCmd.%X0:=false;
	        #OPdwCmd.%X1:=false;
	      ELSE
	       // Automatic mode is not active
	        // Local/Remote mode
	        IF #QREMOTE=false THEN
	          // Local mode is active
	          // OPEN/CLOSE valve by linking (MAN_ON)
	          #QCMD_ON:=#MAN_ON AND NOT #QMAN_AUT;
	          #OPdwCmd.%X0:=false;
	          #OPdwCmd.%X1:=false;
	        ELSE
	         // Remote mode is active
	          // Open valve by operator
	          IF #OPdwCmd.%X1=true THEN
	            #QCMD_ON:=true;
	            #OPdwCmd.%X0:=false;
	            #OPdwCmd.%X1:=false;
	          END_IF;
	          // Close valve by operator
	          IF #OPdwCmd.%X0=true THEN
	            #QCMD_ON:=false;
	            #OPdwCmd.%X0:=false;
	            #OPdwCmd.%X1:=false;
	          END_IF;
	        END_IF;
	      END_IF;
	    ELSE
	      // Local/Remote mode
	      IF #QREMOTE=false THEN
	        // Local mode is active
	          // OPEN/CLOSE valve by linking (SIM_ON)
	          #QCMD_SIM:=#SIM_ON;
	          #OPdwCmd.%X0:=false;
	          #OPdwCmd.%X1:=false;
	      ELSE
	        // Remote mode is active
	          // Open valve by operator
	          IF #OPdwCmd.%X1=true THEN
	            #QCMD_SIM:=true;
	            #OPdwCmd.%X0:=false;
	            #OPdwCmd.%X1:=false;
	          END_IF;
	          // Close valve by operator
	          IF #OPdwCmd.%X0=true THEN
	            #QCMD_SIM:=false;
	            #OPdwCmd.%X0:=false;
	            #OPdwCmd.%X1:=false;
	          END_IF;        
	       END_IF;
	    END_IF;  
	  ELSE
	    // Errors occurs
	    #QCMD_ON:=false;
	    #QCMD_SIM:=false;
	    #OPdwCmd.%X0:=false;
	    #OPdwCmd.%X1:=false;
	  END_IF;
	  
	  (****************************************
	    Network 7: Drive FB_Run
	  *****************************************)
	  #Drive_FB_ON := #IN_SW.%X2 OR ((#IN_SP_Speed < 5.0)AND #QCMD_ON);
	  #QFB_RUN := (#FB_MODE = FALSE AND #Drive_FB_ON) OR (#FB_MODE = TRUE AND (#FB_ON OR ((#IN_SP_Speed < 5.0)AND #QCMD_ON)));
	  (****************************************
	    Network 8: Control signal to the Motor (HMI Status)
	  *****************************************)
	  IF #QERR=false THEN
	    // Motor is stopped
	    IF (((#QFB_RUN=false OR #QMON=false) AND #QSIM=false AND #QCMD_ON=false) OR
	      ((#FB_SIM=false OR #QMON=false) AND #QSIM=true AND #QCMD_SIM=false)) AND #QSTOPPING=true THEN
	      #QSTOP:=true;
	      #QSTOPPING:=false;
	      #QRUN:=false;
	      #QSTARTING:=false;
	      #QwState:=0;
	    END_IF;
	    // Motor is stopping
	    IF ((#QSIM=false AND #QCMD_ON=false) OR (#QSIM=true AND #QCMD_SIM=false)) AND (#QRUN=true OR #QSTARTING=true) THEN
	      #QSTOP:=false;
	      #QSTOPPING:=true;
	      #QRUN:=false;
	      #QSTARTING:=false;
	      #QwState:=3;
	    END_IF;
	    // Motor is running 
	    IF (((#QFB_RUN=true OR #QMON=false) AND #QSIM=false AND #QCMD_ON=true) OR
	      ((#FB_SIM=true OR #QMON=false) AND #QSIM=true AND #QCMD_SIM=true)) AND #QSTARTING=true THEN    
	    #QSTOP:=false;
	    #QSTOPPING:=false;
	    #QRUN:=true;
	    #QSTARTING:=false;
	    #QwState:=2;
	    END_IF;
	    // Motor is starting 
	    IF ((#QSIM=false AND #QCMD_ON=true) OR (#QSIM=true AND #QCMD_SIM=true)) AND #QSTOP=true THEN
	    #QSTOP:=false;
	    #QSTOPPING:=false;
	    #QRUN:=false;
	    #QSTARTING:=true;
	    #QwState:=1;
	    END_IF;
	  END_IF;
	  (*******************************************************************
	    Network 9: Drive Control Word
	    *******************************************************************)
	  //Enable PLC Control
	  #Q_CW.%X1 := true;
	  #Q_CW.%X2 := true;
	  #Q_CW.%X3 := true;
	  #Q_CW.%X4 := true;
	  #Q_CW.%X5 := true;
	  #Q_CW.%X6 := true;
	  #Q_CW.%X10 := true;
	  #Q_CW.%X8 := false;
	  #Q_CW.%X9 := false;
	  #Q_CW.%X12 := false;
	  #Q_CW.%X13 := false;
	  #Q_CW.%X14 := false;
	  #Q_CW.%X15 := false;
	  //Drive ON/OFF
	  IF #QCMD_ON = true THEN
	      #Q_CW.%X0 := true;
	  ELSIF #QCMD_ON = FALSE THEN
	      #Q_CW.%X0 := FALSE;
	  END_IF;
	  //Drive Reversing
	  IF #drive_reversing = true THEN
	  #Q_CW.%X11 := true;
	  ELSIF  #drive_reversing = FALSE THEN
	    #Q_CW.%X11 := FALSE;
	  END_IF;
	//Drive Fault Reset
	  IF #OP_RESET = true THEN
	      #Q_CW.%X7 := true;
	  ELSIF #OP_RESET = FALSE THEN
	      #Q_CW.%X7 := FALSE;
	  END_IF;
	  (*******************************************************************
	    Network 10: Feedbacks for Running monitoring in process and simulation mode
	  ********************************************************************)
	  IF #QSIM=false AND #QMON=true  THEN
	  // Feedback monitoring in process mode
	    #TSTARTING(IN:=#QSTARTING,
	               PT:=#MON_T,
	               Q=>#MON_ERR_STARTING,
	               ET=>#QMON_T);
	     
	    #TSTOPPING(IN:=#QSTOPPING,
	              PT:=#MON_T_STOP,
	              Q=>#MON_ERR_STOPPING,
	              ET=>#QMON_T_STOP);
	    // Feedback error
	   #FB_ERR := (#QRUN AND NOT #QFB_RUN) OR (#QSTOP AND #QFB_RUN);
	    IF #FB_ERR=true OR #MON_ERR_STARTING=true OR #MON_ERR_STOPPING=true THEN
	      #QMON_ERR:=true;
	    END_IF;
	    
	    
	  ELSIF #QSIM=true AND #QMON=true THEN
	    // Feedback monitoring in simulation mode
	    #TSTARTING_SIM(IN:=#QSTARTING,
	                  PT:=#SIM_T,
	                  Q=>#MON_SIM_STARTING,
	                  ET=>#QSIM_T);
	    
	    #TSTOPPING_SIM(IN:=#QSTOPPING,
	                  PT:=#SIM_T_STOP,
	                  Q=>#MON_SIM_STOPPING,
	                  ET=>#QSIM_T_STOP);
	    
	    // Feedback for start/stop motor in simulation mode
	    IF #MON_SIM_STOPPING=true OR #QERR=true THEN
	      // Feedback for stop
	      #FB_SIM:=false;
	    ELSIF #MON_SIM_STARTING=true THEN
	      // Feedback for start
	      #FB_SIM:=true;
	    END_IF;
	  END_IF;
	
	  (*******************************************************************
	    Network 11: Feedbacks for flow monitoring in process and simulation mode
	  ********************************************************************)
	// Delay time for feedbak flow monitoring
	  #START_FLOW_TIME:=#QFLOW_MON AND (#QSTARTING OR #QRUN) AND NOT #QFLOW_MON_ACK;
	  #TFLOW(IN:=#START_FLOW_TIME,
	         PT:=#FLOW_MT,
	         Q=>#MON_ERR_FLOW,
	         ET=>#QFLOW_MT);
	  
	  //
	  #START_FLOW_TIME2:=false;
	  IF (#FLOW < #FLOW_LL) THEN
	    #START_FLOW_TIME2:=true;
	  END_IF;
	  
	     #TFLOW(IN:=#START_FLOW_TIME2,
	         PT:=#FLOW_MT,
	         Q=>#MON_ERR_FLOW2,
	         ET=>#QFLOW_MT);
	   IF #MON_ERR_FLOW2 THEN
	      #QFLOW_ERR:=true;
	   END_IF;
	  (**********************************************
	    Network 12: Drive Set Speed
	   ***********************************************)
	   //Drive Setpoint Speed in Hz
	   #SP_SpeedHz := #IN_SP_Speed / 2;
	   //Limit Speed 0 to 50 Hz
	   IF #SP_SpeedHz<0.0 THEN
	       GOTO N004;
	   END_IF;
	   IF #SP_SpeedHz > 50.0 THEN
	        GOTO N004;
	    END_IF;
	//OUT = [ ((IN–LO_LIM)/(HI_LIM–LO_LIM)) ∗ (K2–K1) ] + K1
	//UNSCALE Setpoint Speed VSD with hardwire
	//#Q_SP := REAL_TO_INT(((((#IN_SP / 2) - #SP_Lo) / (#SP_Hi - #SP_Lo)) * (#SP_K2 - #SP_K1)) + #SP_K1);
	    IF #FB_MODE = TRUE THEN
	        #Q_SP_Speed := DINT_TO_WORD(ROUND(#SP_SpeedHz * real#100.0) * DINT#27648 / DINT#5000);
	        #Drive_Actual_Speed := (INT_TO_REAL(#"IN _AV") / 27648.0 * 100.0);
	    ELSIF #FB_MODE = FALSE THEN
	        #Q_SP_Speed := DINT_TO_WORD(ROUND(#SP_SpeedHz * real#100.0) * DINT#16384 / DINT#5000);
	        #Drive_Actual_Speed := (INT_TO_REAL(#"IN _AV") / 16354.0 * 100.0);
	    END_IF;
	N004:  ;
	    
	   (**********************************************
	    Network 13: Drive Actual
	  ***********************************************)
	    #QAct_Speed := #Drive_Actual_Speed;
	//    #QAct_Volt := (INT_TO_REAL(#IN_Volt) / 16354.0 * 1000.0);
	//    #QAct_Amp := (INT_TO_REAL(#IN_Ampere) / 16354.0 * 100.0);
	//    #QAct_KW := (INT_TO_REAL(#IN_KW) / 16354.0 * 100.0);
	//    #QAct_Nm := (INT_TO_REAL(#IN_Nm) / 16354.0 * 100.0);
	  (**********************************************
	    Network 14: Check errors
	  ***********************************************)
	   //Drive Fault
	   #QDrive_Fault := #IN_SW.%X3;
	   //Drive Alarm
	   #QDrive_Alarm := #IN_SW.%X7;
	   // External error
	  #QERR_EXT:=#ERR_EXTERN;  
	  // Interlock error
	  IF #LOCK=true AND ( #QSTARTING=true OR #QRUN=true) THEN
	    #QLOCK:=true;
	  END_IF;
	  //
	  IF #MPS=true THEN
	    #QMPS:=true;
	  END_IF;
	  
	  // Error in valve condition
	  #CON_ERR:=NOT((#QSTOP AND NOT #QSTARTING AND NOT #QRUN AND NOT #QSTOPPING) OR
	  (NOT #QSTOP AND #QSTARTING AND NOT #QRUN AND NOT #QSTOPPING) OR
	  (NOT #QSTOP AND NOT #QSTARTING AND #QRUN AND NOT #QSTOPPING) OR
	  (NOT #QSTOP AND NOT #QSTARTING AND NOT #QRUN AND #QSTOPPING));
	
	  (**********************************************
	    Network 15: General error
	  ***********************************************)
	  #QERR:=#QDrive_Fault OR #QDrive_Alarm OR #QERR_EXT OR #QMON_ERR OR #QFLOW_ERR OR #QMPS OR #QLOCK OR #CON_ERR;
	  
	  (**********************************************
	    Network 16: If error then stop
	  ***********************************************)
	  IF #QERR=true THEN
	    #QSTOP:=true;
	    #QSTARTING:=false;
	    #QRUN:=false;
	    #QSTOPPING:=false;
	    #QwState:=0;
	  END_IF;
	  // Reset errors
	  IF #OP_RESET=true THEN
	    #QMON_ERR:=false;
	    #QLOCK:=false;
	    #QFLOW_ERR:=false;
	    #QMPS:=false;
	  END_IF;
	    // End normal case
	END_IF;
	
	(****************************************************
	  Network 13: Influence visibility of faceplate window
	*****************************************************)
	IF #OP_VISIBILITY<>#VISIBILITY_OLD THEN
	  #VISIBILITY_OLD:=#OP_VISIBILITY;
	  #VISIBILITY:=#OP_VISIBILITY;
	ELSIF #VISIBILITY<>#VISIBILITY_OLD THEN
	  #VISIBILITY_OLD:=#VISIBILITY;
	  #OP_VISIBILITY:=#VISIBILITY;
	END_IF;
	(********************************
	  Network 14: Set state for HMI
	*********************************)
	#QdwState.%X0:=#QSTOP AND NOT #QERR;
	#QdwState.%X1:=#QSTARTING;
	#QdwState.%X2:=#QRUN;
	#QdwState.%X3:=#QSTOPPING;
	#QdwState.%X4:=false;
	#QdwState.%X5:=false;
	#QdwState.%X6:=false;
	#QdwState.%X7:=false;
	#QdwState.%X8:=#QMON;
	#QdwState.%X9:=#QMON_ERR;
	#QdwState.%X10:=#QFLOW_MON;
	#QdwState.%X11:=#QFLOW_ERR;
	#QdwState.%X12:=#QMPS;
	#QdwState.%X13:=#QDrive_Fault;
	#QdwState.%X14:=#QDrive_Alarm;
	#QdwState.%X15:=false;
	#QdwState.%X16:=#QMAN_AUT;
	#QdwState.%X17:=#QREMOTE;
	#QdwState.%X18:=#QSIM;
	#QdwState.%X19:=false;
	#QdwState.%X20:=false;
	#QdwState.%X21:=false;
	#QdwState.%X22:=false;
	#QdwState.%X23:=false;
	#QdwState.%X24:=#QERR;
	#QdwState.%X25:=#QERR_EXT;
	#QdwState.%X26:=#QLOCK;
	#QdwState.%X27:=#LOCK;
	#QdwState.%X28:=false;
	#QdwState.%X29:=false;
	#QdwState.%X30:=false;
	#QdwState.%X31:=false;
	
	(********************************
	  Network 15: Bit alarm procedure
	*********************************)
	#QwAlarm.%X0:=#QMON_ERR;
	#QwAlarm.%X1:=#QFLOW_ERR;
	#QwAlarm.%X2:=#MPS;
	#QwAlarm.%X3:=#QDrive_Fault;
	#QwAlarm.%X4:=#QLOCK;
	#QwAlarm.%X5:=#QDrive_Alarm;
	#QwAlarm.%X6:=#QERR_EXT;
	#QwAlarm.%X7:=#QERR;
	#QwAlarm.%X8:=#QSTOP;
	#QwAlarm.%X9:=#QSTARTING;
	#QwAlarm.%X10:=#QRUN;
	#QwAlarm.%X11:=#QSTOPPING;
	#QwAlarm.%X12:=#LOCK;
	#QwAlarm.%X13:=#QREMOTE;
	#QwAlarm.%X14:=#QMAN_AUT;
	#QwAlarm.%X15:=#QSIM;
END_FUNCTION_BLOCK

FUNCTION_BLOCK "PIDCtrlV2"
{ S7_Optimized_Access := 'FALSE' }
NAME : PIDCtrl
VERSION : 1.0
   VAR_INPUT 
      InvertControl : Bool := 0;   // Enables inversion of control logic
      InputPerOn : Bool := 0;   // Selection of process value
      InputUpperLimit : Real := 120.0;   // Entry for process value high limit
      InputLowerLimit : Real := 0.0;   // Entry for process value low limit
      UpperPointOut : Real := 100.0;   // Entry for scaled high process value
      LowerPointOut : Real := 0.0;   // Entry for scaled low process value
      UpperPointIn : Real := 27648.0;   // Entry for high value of Input_PER
      LowerPointIn : Real := 0.0;   // Entry for low value of Input_PER
      InputUpperWarning : Real := 200.0;   // Entry for warning high limit
      InputLowerWarning : Real := -200.0;   // Entry for warning low limit
      MinimumOnTime : Real := 0.0;   // Entry for minimum ON time
      MinimumOffTime : Real := 0.0;   // Entry for minimum OFF time
      OutputUpperLimit : Real := 100.0;   // Entry for high limit of output value
      OutputLowerLimit : Real := 0.0;   // Entry for low limit of output value
      SetpointUpperLimit : Real := 100.0;   // High limit of setpoint
      SetpointLowerLimit : Real := 0.0;   // Low limit of the setpoint
      PIDManualEnable : Bool := 0;   // Enables manual entry of PID parameters
      Gain : Real := 1.0;   // Entry for proportional gain
      Ti : Real := 20.0;   // Entry for integral action time
      Td : Real := 0.0;   // Entry for derivative action time
      TdFiltRatio : Real := 0.0;   // Entry for derivative delay coefficient
      PWeighting : Real := 1.0;   // Entry for proportional action weighting
      DWeighting : Real := 1.0;   // Entry for derivative action weighting
      Cycle : Real := 0.5;   // Entry for sampling time for the PID algorithm
      Setpoint : Real := 0.0;   // Setpoint of the PID controller in automatic mode
      Input : Real := 0.0;   // Process value in REAL format
      Input_PER : Int := 0;   // Analog process value
      ManualValue : Real := 0.0;   // This value is used as the output value in manual mode
      LOCK : Bool := 0;   // 1 = Interlock active
      ERR_EXTERN : Bool := 0;   // 1 = External error arised
      LIOP_SEL : Bool := 0;   // 0 = Operator; 1 = Linking
      L_AUT : Bool := 1;   // 0 = Manual; 1 = Automatic
      L_REMOTE : Bool := 0;   // 0 = Local; 1 = Remote
      L_RESET : Bool := 0;   // 1 = Reset error peripherie
      INSTANCE : String[254] := 'PIDCtrlV2_001';   // Filter attribute for message view, also used for labelling
      RESTART : Bool := 0;   // 1 = Initialize FB at startup (first cycle of PLC)
   END_VAR

   VAR_OUTPUT 
      QSetpoint : Real := 0.0;   // Setpoint of the PID controller
      ScaledInput : Real := 0.0;   // Scaled process value
      Output : Real := 0.0;   // Output value in REAL format
      Output_PER : Int := 0;   // Analog output value
      Output_PWM : Bool := 0;   // 1 = Pulse-width-modulated output value active
      SetpointLimit_H : Bool := 0;   // 1 = Setpoint absolute high limit has been reached
      SetpointLimit_L : Bool := 0;   // 1 = Setpoint absolute low limit has been reached
      InputWarning_H : Bool := 0;   // 1 = Process value has been reached or exceeded the warning high limit
      InputWarning_L : Bool := 0;   // 1 = Process value has been reached or fallen below the warning low limit
      State : Int := 0;   // Current operating mode of the PID controller
      Error : Bool := 0;   // 1 = at least one error message is pending in this cycle
      ErrorBits : DWord := 16#00000000;   // This parameter shows which error messages are pending
      QGain : Real := 0.0;   // Setpoint of proportional gain
      QTi : Real := 0.0;   // Setpoint of integral action time
      QTd : Real := 0.0;   // Setpoint of derivative action time
      QdwState : DWord := 16#00000000;   // Status HMI
      QPERIPH : Bool := 0;   // 1 = Analog process value active
      QMAN_AUT : Bool := 0;   // 0 = Manual; 1 = Process
      QREMOTE : Bool := 0;   // 0 = Local; 1 = Remote
      QLOCK : Bool := 0;   // 1 = Interlock is active
      QERR : Bool := 0;   // 1 = Common error
      QERR_EXT : Bool := 0;   // 1 = External error
      QwAlarm : Word := 16#0000;   // Bit alarm procedure
   END_VAR

   VAR_IN_OUT 
      VISIBILITY : Word := 16#0000;   // Bit 0: Tab1 of window; Bit 1: Tab2 of window; ... ; Bit 7: Minimize
      OPdwCmd : DWord := 16#00000000;   // Contorl word HMI
   END_VAR

   VAR 
      OP_Input_PER_On : Bool := 0;
      OP_Setpoint : Real := 0.0;
      OP_Output : Real := 0.0;
      OP_ManualValue : Real := 0.0;
      OP_InvertControl : Bool := 0;
      OP_Cycle : Real := 0.0;
      OP_Gain : Real := 0.0;
      OP_Ti : Real := 0.0;
      OP_Td : Real := 0.0;
      OP_TdFiltRatio : Real := 0.0;
      OP_PWeighting : Real := 0.0;
      OP_DWeighting : Real := 0.0;
      OP_OutputUpperLimit : Real := 100.0;
      OP_OutputLowerLimit : Real := 0.0;
      OP_MinimumOnTime : Real := 0.0;
      OP_MinimumOffTime : Real := 0.0;
      OP_SetpointUpperLimit : Real := 0.0;
      OP_SetpointLowerLimit : Real := 0.0;
      OP_InputUpperLimit : Real := 0.0;
      OP_InputLowerLimit : Real := 0.0;
      OP_LowerPointIn : Real := 0.0;
      OP_UpperPointIn : Real := 0.0;
      OP_LowerPointOut : Real := 0.0;
      OP_UpperPointOut : Real := 0.0;
      OP_InputUpperWarning : Real := 0.0;
      OP_InputLowerWarning : Real := 0.0;
      OP_State : Int := 0;
      OP_VISIBILITY : Word := 16#0000;
      VISIBILITY_OLD : Word := 16#0000;
      TP_SEL : Bool := 0;
      TI_SEL : Bool := 0;
      TD_SEL : Bool := 0;
      ManualEnable : Bool;
      ERR_EXTERN_OLD : Bool;
      L_RESET_OLD : Bool;
   END_VAR


BEGIN
	// Start up
	IF #RESTART THEN // Restart case   
	  #VISIBILITY := W#16#0;
	ELSE // Normal case
	    
	  // Check errors ===========================================================
	  #QERR_EXT := #ERR_EXTERN; // 1 = External error
	  #QLOCK := #LOCK; // 1 = Interlock is active
	  
	  IF (#ERR_EXTERN AND NOT #ERR_EXTERN_OLD) THEN
	      #QERR := TRUE;
	  END_IF;
	  
	  // MANUAL/PROCESS Operation ===============================================
	  IF ((#LIOP_SEL AND NOT #L_AUT) OR (#OPdwCmd.%X16 AND NOT #LIOP_SEL)) THEN
	      #QMAN_AUT := FALSE; // 0 = Manual
	  ELSIF ((#LIOP_SEL AND #L_AUT) OR (#OPdwCmd.%X17 AND NOT #LIOP_SEL)) THEN
	      #QMAN_AUT := TRUE; // 1 = Process
	  END_IF;
	    
	  IF NOT #QLOCK THEN
	      #ManualEnable := NOT #QMAN_AUT;
	  END_IF;
	  
	  // LOCAL/REMOTE Operation =================================================
	  IF ((#LIOP_SEL AND NOT #L_REMOTE) OR (#OPdwCmd.%X18 AND NOT #LIOP_SEL)) THEN
	      #QREMOTE := FALSE; // 0 = Local
	  ELSIF ((#LIOP_SEL AND #L_REMOTE) OR (#OPdwCmd.%X19 AND NOT #LIOP_SEL)) THEN
	      #QREMOTE := TRUE; // 1 = Remote
	  END_IF;
	      
	  // Toggle Invert Control ==================================================
	  IF (#OPdwCmd.%X5 AND NOT #LIOP_SEL AND #QREMOTE AND NOT #QLOCK) THEN
	      #OP_InvertControl := NOT #OP_InvertControl;
	  END_IF;
	      
	  // SET Periphery/Extern connection ========================================
	  IF (NOT #InputPerOn AND NOT #QREMOTE AND NOT #QLOCK) OR (#OPdwCmd.%X7 AND #QREMOTE AND NOT #QLOCK) THEN
	      #QPERIPH := FALSE; // 0 = Extern
	  ELSIF (#InputPerOn AND NOT #QREMOTE AND NOT #QLOCK) OR (#OPdwCmd.%X6 AND #QREMOTE AND NOT #QLOCK) THEN
	    #QPERIPH := TRUE; // 1 = Periphery
	  END_IF;
	 
	  // Initialization of the PID Parameter ====================================
	  IF (NOT #QLOCK AND NOT #QREMOTE) THEN // Local control (PIDCtrlV2 Input)
	    
	    "PID_Compact_1".Config.InvertControl              := #InvertControl;
	    "PID_Compact_1".Config.InputPerOn                 := #QPERIPH;
	    "PID_Compact_1".Config.InputUpperLimit            := #InputUpperLimit;
	    "PID_Compact_1".Config.InputLowerLimit            := #InputLowerLimit;
	    "PID_Compact_1".Config.InputScaling.UpperPointOut := #UpperPointOut;
	    "PID_Compact_1".Config.InputScaling.LowerPointOut := #LowerPointOut;
	    "PID_Compact_1".Config.InputScaling.UpperPointIn  := #UpperPointIn;
	    "PID_Compact_1".Config.InputScaling.LowerPointIn  := #LowerPointIn;
	    "PID_Compact_1".Config.InputUpperWarning          := #InputUpperWarning;
	    "PID_Compact_1".Config.InputLowerWarning          := #InputLowerWarning;
	    "PID_Compact_1".Config.MinimumOnTime              := #MinimumOnTime;
	    "PID_Compact_1".Config.MinimumOffTime             := #MinimumOffTime;
	    "PID_Compact_1".Config.OutputUpperLimit           := #OutputUpperLimit;
	    "PID_Compact_1".Config.OutputLowerLimit           := #OutputLowerLimit;
	    "PID_Compact_1".Config.SetpointUpperLimit         := #SetpointUpperLimit;
	    "PID_Compact_1".Config.SetpointLowerLimit         := #SetpointLowerLimit;
	    
	    IF #PIDManualEnable THEN // Manual parameter setting release
	      
	      "PID_Compact_1".Retain.CtrlParams.Gain        := #Gain;
	      "PID_Compact_1".Retain.CtrlParams.Ti          := #Ti;
	      "PID_Compact_1".Retain.CtrlParams.Td          := #Td;
	      "PID_Compact_1".Retain.CtrlParams.TdFiltRatio := #TdFiltRatio;
	      "PID_Compact_1".Retain.CtrlParams.PWeighting  := #PWeighting;
	      "PID_Compact_1".Retain.CtrlParams.DWeighting  := #DWeighting;
	      "PID_Compact_1".Retain.CtrlParams.Cycle       := #Cycle;
	      
	  END_IF;
	    
	    #OP_Setpoint := #Setpoint;
	    #OP_ManualValue := #ManualValue;
	    
	  ELSIF (NOT #QLOCK AND #QREMOTE) THEN // Remote control (HMI)
	      
	    "PID_Compact_1".Config.InvertControl              := #OP_InvertControl;
	    "PID_Compact_1".Config.InputPerOn                 := #QPERIPH;
	    "PID_Compact_1".Config.InputUpperLimit            := #OP_InputUpperLimit;
	    "PID_Compact_1".Config.InputLowerLimit            := #OP_InputLowerLimit;
	    "PID_Compact_1".Config.InputScaling.UpperPointOut := #OP_UpperPointOut;
	    "PID_Compact_1".Config.InputScaling.LowerPointOut := #OP_LowerPointOut;
	    "PID_Compact_1".Config.InputScaling.UpperPointIn  := #OP_UpperPointIn;
	    "PID_Compact_1".Config.InputScaling.LowerPointIn  := #OP_LowerPointIn;
	    "PID_Compact_1".Config.InputUpperWarning          := #OP_InputUpperWarning;
	    "PID_Compact_1".Config.InputLowerWarning          := #OP_InputLowerWarning;
	    "PID_Compact_1".Config.MinimumOnTime              := #OP_MinimumOnTime;
	    "PID_Compact_1".Config.MinimumOffTime             := #OP_MinimumOffTime;
	    "PID_Compact_1".Config.OutputUpperLimit           := #OP_OutputUpperLimit;
	    "PID_Compact_1".Config.OutputLowerLimit           := #OP_OutputLowerLimit;
	    "PID_Compact_1".Config.SetpointUpperLimit         := #OP_SetpointUpperLimit;
	    "PID_Compact_1".Config.SetpointLowerLimit         := #OP_SetpointLowerLimit;
	    
	    "PID_Compact_1".Retain.CtrlParams.Gain            := #OP_Gain;
	    "PID_Compact_1".Retain.CtrlParams.Ti              := #OP_Ti;
	    "PID_Compact_1".Retain.CtrlParams.Td              := #OP_Td;
	    "PID_Compact_1".Retain.CtrlParams.TdFiltRatio     := #OP_TdFiltRatio;
	    "PID_Compact_1".Retain.CtrlParams.PWeighting      := #OP_PWeighting;
	    "PID_Compact_1".Retain.CtrlParams.DWeighting      := #OP_DWeighting;
	    "PID_Compact_1".Retain.CtrlParams.Cycle           := #OP_Cycle;
	
	  END_IF;
	  
	  // Call PID_Compact V2 ====================================================  
	  "PID_Compact_1"
	    (
	        Setpoint        := #OP_Setpoint,
	        Input           := #Input,
	        Input_PER       := #Input_PER,
	        ManualEnable    := #ManualEnable,
	        ManualValue     := #OP_ManualValue,
	        Reset           := #OPdwCmd.%X24,
	        ScaledInput     => #ScaledInput,
	        Output          => #Output,
	        Output_PER      => #Output_PER,
	        Output_PWM      => #Output_PWM,
	        SetpointLimit_H => #SetpointLimit_H,
	        SetpointLimit_L => #SetpointLimit_L,
	        InputWarning_H  => #InputWarning_H,
	        InputWarning_L  => #InputWarning_L,
	        State           => #State,
	        Error           => #Error,
	        ErrorBits       => #ErrorBits
	    );
	  
	  // Tuning values ==========================================================
	  #OP_State              := #State;
	  #OP_Input_PER_On       := "PID_Compact_1".Config.InputPerOn;
	  #OP_Setpoint           := "PID_Compact_1".Setpoint;
	  #QSetpoint             := #OP_Setpoint;
	  #OP_Output             := "PID_Compact_1".Output;
	  #OP_ManualValue        := "PID_Compact_1".ManualValue;
	  #OP_InvertControl      := "PID_Compact_1".Config.InvertControl;
	  
	  // Scaling values for Input_PER ===========================================
	  #OP_LowerPointIn       := "PID_Compact_1".Config.InputScaling.LowerPointIn;
	  #OP_UpperPointIn       := "PID_Compact_1".Config.InputScaling.UpperPointIn;
	  
	  // Limits for scaled process value ========================================
	  #OP_LowerPointOut      := "PID_Compact_1".Config.InputScaling.LowerPointOut;
	  #OP_UpperPointOut      := "PID_Compact_1".Config.InputScaling.UpperPointOut;
	  
	  // Setpoint value limits ==================================================
	  #OP_SetpointUpperLimit := "PID_Compact_1".Config.SetpointUpperLimit;
	  #OP_SetpointLowerLimit := "PID_Compact_1".Config.SetpointLowerLimit;
	  
	  // Actual value limits ====================================================
	  #OP_InputUpperLimit    := "PID_Compact_1".Config.InputUpperLimit;
	  #OP_InputLowerLimit    := "PID_Compact_1".Config.InputLowerLimit;
	  #OP_InputUpperWarning  := "PID_Compact_1".Config.InputUpperWarning;
	  #OP_InputLowerWarning  := "PID_Compact_1".Config.InputLowerWarning;
	  
	  // Output value limits ====================================================
	  #OP_OutputUpperLimit   := "PID_Compact_1".Config.OutputUpperLimit;
	  #OP_OutputLowerLimit   := "PID_Compact_1".Config.OutputLowerLimit;
	  
	  // PWM value limits =======================================================
	  #OP_MinimumOnTime      := "PID_Compact_1".Config.MinimumOnTime;
	  #OP_MinimumOffTime     := "PID_Compact_1".Config.MinimumOffTime;
	  
	  // Control parameters =====================================================
	  #OP_Gain               := "PID_Compact_1".Retain.CtrlParams.Gain;
	  #QGain                 := #OP_Gain;
	  #OP_Ti                 := "PID_Compact_1".Retain.CtrlParams.Ti;
	  #QTi                   := #OP_Ti;
	  #OP_Td                 := "PID_Compact_1".Retain.CtrlParams.Td;
	  #QTd                   := #OP_Td;
	  #OP_TdFiltRatio        := "PID_Compact_1".Retain.CtrlParams.TdFiltRatio;
	  #OP_PWeighting         := "PID_Compact_1".Retain.CtrlParams.PWeighting;
	  #OP_DWeighting         := "PID_Compact_1".Retain.CtrlParams.DWeighting;
	  #OP_Cycle              := "PID_Compact_1".Retain.CtrlParams.Cycle;
	  
	  // P action ===============================================================
	  IF (#OP_Gain > 0.0) THEN
	    #TP_SEL := TRUE;
	  ELSE
	    #TP_SEL := FALSE;
	  END_IF;
	  
	  // I action ===============================================================
	  IF (#OP_Ti > 0.0) THEN
	    #TI_SEL := TRUE;
	  ELSE
	    #TI_SEL := FALSE;
	  END_IF;
	  
	  // D action ===============================================================
	  IF (#OP_Td > 0.0) THEN
	    #TD_SEL := TRUE;
	  ELSE
	    #TD_SEL := FALSE;
	  END_IF;
	  
	  // Set visibility of faceplate ============================================
	  IF (#OP_VISIBILITY <> #VISIBILITY_OLD) THEN
	    #VISIBILITY_OLD := #OP_VISIBILITY;
	    #VISIBILITY := #OP_VISIBILITY;
	  ELSIF (#VISIBILITY <> #VISIBILITY_OLD) THEN
	    #VISIBILITY_OLD := #VISIBILITY;
	    #OP_VISIBILITY := #VISIBILITY;
	  END_IF;
	  
	  // Reset error ============================================================
	  IF (((#OPdwCmd.%X24 AND #QREMOTE) OR (#L_RESET AND NOT #L_RESET_OLD)) AND NOT #ERR_EXTERN) THEN
	      #QERR := FALSE;
	  END_IF;
	  
	  // Save signals for edge detect ===========================================
	  #L_RESET_OLD := #L_RESET;
	  #ERR_EXTERN_OLD := #ERR_EXTERN;
	  
	  // Reset commands =========================================================
	  #OPdwCmd := DW#16#0;
	  
	  // Set state for HMI ======================================================
	  #QdwState.%X0  := #TP_SEL;
	  #QdwState.%X1  := #TI_SEL;
	  #QdwState.%X2  := #TD_SEL;
	  #QdwState.%X3  := FALSE;
	  #QdwState.%X4  := FALSE;
	  #QdwState.%X5  := #OP_InvertControl;
	  #QdwState.%X6  := #QPERIPH;
	  #QdwState.%X7  := FALSE;
	  #QdwState.%X8  := FALSE;
	  #QdwState.%X9  := FALSE;
	  #QdwState.%X10 := FALSE;
	  #QdwState.%X11 := FALSE;
	  #QdwState.%X12 := #SetpointLimit_L;
	  #QdwState.%X13 := #InputWarning_L AND NOT #SetpointLimit_L;
	  #QdwState.%X14 := #InputWarning_H AND NOT #SetpointLimit_H;
	  #QdwState.%X15 := #SetpointLimit_H;
	  #QdwState.%X16 := #QMAN_AUT;
	  #QdwState.%X17 := #QREMOTE;
	  #QdwState.%X18 := FALSE;
	  #QdwState.%X19 := FALSE;
	  #QdwState.%X20 := FALSE;
	  #QdwState.%X21 := FALSE;
	  #QdwState.%X22 := FALSE;
	  #QdwState.%X23 := FALSE;
	  #QdwState.%X24 := #QERR;
	  #QdwState.%X25 := #QERR_EXT;
	  #QdwState.%X26 := #QLOCK;
	  #QdwState.%X27 := #LOCK;
	  #QdwState.%X28 := FALSE;
	  #QdwState.%X29 := FALSE;
	  #QdwState.%X30 := FALSE;
	  #QdwState.%X31 := FALSE;
	  
	  // Bit alarm procedure ====================================================
	  #QwAlarm.%X0  := #SetpointLimit_L;
	  #QwAlarm.%X1  := #SetpointLimit_H;
	  #QwAlarm.%X2  := FALSE;
	  #QwAlarm.%X3  := FALSE;
	  #QwAlarm.%X4  := #QLOCK;
	  #QwAlarm.%X5  := FALSE;
	  #QwAlarm.%X6  := #QERR_EXT;
	  #QwAlarm.%X7  := #QERR;
	  #QwAlarm.%X8  := #InputWarning_L;
	  #QwAlarm.%X9  := #InputWarning_H;
	  #QwAlarm.%X10 := NOT #QPERIPH;
	  #QwAlarm.%X11 := #QPERIPH;
	  #QwAlarm.%X12 := NOT #QREMOTE;
	  #QwAlarm.%X13 := #QREMOTE;
	  #QwAlarm.%X14 := NOT #QMAN_AUT;
	  #QwAlarm.%X15 := #QMAN_AUT;
	
	END_IF; // End normal case
END_FUNCTION_BLOCK

DATA_BLOCK "Alarm_Collector_Gen_DB"   // DB65
VERSION : 0.1
// stored: AutoNumber true, DBAccessibleFromOPCUA true, DBAccessibleFromWebserver true, InstanceOfName Alarm_Collector_Gen, InstanceOfType FB
"Alarm_Collector_Gen"
BEGIN
END_DATA_BLOCK

DATA_BLOCK "ReadDateandTime_DB"   // DB31
VERSION : 0.1
// stored: AutoNumber false, DBAccessibleFromOPCUA true, DBAccessibleFromWebserver true, InstanceOfName ReadDateandTime, InstanceOfType FB
"ReadDateandTime"
BEGIN
END_DATA_BLOCK

DATA_BLOCK "Sim_PTM_DB"   // DB1000
VERSION : 0.1
// stored: AutoNumber false, DBAccessibleFromOPCUA true, DBAccessibleFromWebserver true, InstanceOfName Sim_PT1, InstanceOfType FB
"Sim_PT1"
BEGIN
END_DATA_BLOCK

DATA_BLOCK "Sim_PTS_DB"   // DB1001
VERSION : 0.1
// stored: AutoNumber false, DBAccessibleFromOPCUA true, DBAccessibleFromWebserver true, InstanceOfName Sim_PT1, InstanceOfType FB
"Sim_PT1"
BEGIN
END_DATA_BLOCK

DATA_BLOCK "AlarmFlowColletor"   // DB217
VERSION : 0.1
// stored: AutoNumber false, DBAccessibleFromOPCUA true, DBAccessibleFromWebserver true, InstanceOfName Alarm Flow Collector, InstanceOfType FB
"Alarm Flow Collector"
BEGIN
END_DATA_BLOCK

DATA_BLOCK "Blend_T-20"   // DB211
VERSION : 0.1
// stored: AutoNumber false, DBAccessibleFromOPCUA true, DBAccessibleFromWebserver true, InstanceOfName Blend_Tank, InstanceOfType FB
"Blend_Tank"
BEGIN
END_DATA_BLOCK

DATA_BLOCK "Blend_T-21"   // DB212
VERSION : 0.1
// stored: AutoNumber false, DBAccessibleFromOPCUA true, DBAccessibleFromWebserver true, InstanceOfName Blend_Tank, InstanceOfType FB
"Blend_Tank"
BEGIN
END_DATA_BLOCK

DATA_BLOCK "Blend_T-30"   // DB213
VERSION : 0.1
// stored: AutoNumber false, DBAccessibleFromOPCUA true, DBAccessibleFromWebserver true, InstanceOfName Blend_Tank, InstanceOfType FB
"Blend_Tank"
BEGIN
END_DATA_BLOCK

DATA_BLOCK "Blend_T-31"   // DB214
VERSION : 0.1
// stored: AutoNumber false, DBAccessibleFromOPCUA true, DBAccessibleFromWebserver true, InstanceOfName Blend_Tank, InstanceOfType FB
"Blend_Tank"
BEGIN
END_DATA_BLOCK

DATA_BLOCK "Blend_T-40"   // DB215
VERSION : 0.1
// stored: AutoNumber false, DBAccessibleFromOPCUA true, DBAccessibleFromWebserver true, InstanceOfName Blend_Tank, InstanceOfType FB
"Blend_Tank"
BEGIN
END_DATA_BLOCK

DATA_BLOCK "Blend_T-41"   // DB216
VERSION : 0.1
// stored: AutoNumber false, DBAccessibleFromOPCUA true, DBAccessibleFromWebserver true, InstanceOfName Blend_Tank, InstanceOfType FB
"Blend_Tank"
BEGIN
END_DATA_BLOCK

DATA_BLOCK "GetData_DB"   // DB45
AUTHOR : SiemensIndustryOnlineSupport
FAMILY : S7comm
VERSION : 1.0
// stored: AutoNumber true, DBAccessibleFromOPCUA true, DBAccessibleFromWebserver true, InstanceOfName GetData, InstanceOfType FB
"GetData"
BEGIN
END_DATA_BLOCK

DATA_BLOCK "THE1_GetData_DB"   // DB16
AUTHOR : SiemensIndustryOnlineSupport
FAMILY : S7comm
VERSION : 1.0
// stored: AutoNumber true, DBAccessibleFromOPCUA true, DBAccessibleFromWebserver true, InstanceOfName GetData, InstanceOfType FB
"GetData"
BEGIN
END_DATA_BLOCK

DATA_BLOCK "THE2_GetData_DB"   // DB17
AUTHOR : SiemensIndustryOnlineSupport
FAMILY : S7comm
VERSION : 1.0
// stored: AutoNumber true, DBAccessibleFromOPCUA true, DBAccessibleFromWebserver true, InstanceOfName GetData, InstanceOfType FB
"GetData"
BEGIN
END_DATA_BLOCK

DATA_BLOCK "T-12.00_Homomixer"   // DB102
VERSION : 0.1
// stored: AutoNumber false, DBAccessibleFromOPCUA true, DBAccessibleFromWebserver true, InstanceOfName Homomix, InstanceOfType FB
"Homomix"
BEGIN
END_DATA_BLOCK

DATA_BLOCK "T-13.00_Homomixer"   // DB103
VERSION : 0.1
// stored: AutoNumber false, DBAccessibleFromOPCUA true, DBAccessibleFromWebserver true, InstanceOfName Homomix, InstanceOfType FB
"Homomix"
BEGIN
END_DATA_BLOCK

DATA_BLOCK "T-14.00_Homomixer"   // DB104
VERSION : 0.1
// stored: AutoNumber false, DBAccessibleFromOPCUA true, DBAccessibleFromWebserver true, InstanceOfName Homomix, InstanceOfType FB
"Homomix"
BEGIN
END_DATA_BLOCK

DATA_BLOCK "T-23.00"   // DB37
VERSION : 0.1
// stored: AutoNumber false, DBAccessibleFromOPCUA true, DBAccessibleFromWebserver true, InstanceOfName Storage_Tank_Multi_Inload, InstanceOfType FB
"Storage_Tank_Multi_Inload"
BEGIN
END_DATA_BLOCK

DATA_BLOCK "T-24.00"   // DB55
VERSION : 0.1
// stored: AutoNumber false, DBAccessibleFromOPCUA true, DBAccessibleFromWebserver true, InstanceOfName Storage_Tank_Multi_Inload, InstanceOfType FB
"Storage_Tank_Multi_Inload"
BEGIN
END_DATA_BLOCK

DATA_BLOCK "T-29.00"   // DB38
VERSION : 0.1
// stored: AutoNumber true, DBAccessibleFromOPCUA true, DBAccessibleFromWebserver true, InstanceOfName Storage_Tank_Single_Inload, InstanceOfType FB
"Storage_Tank_Single_Inload"
BEGIN
END_DATA_BLOCK

DATA_BLOCK "T-33.00"   // DB41
VERSION : 0.1
// stored: AutoNumber false, DBAccessibleFromOPCUA true, DBAccessibleFromWebserver true, InstanceOfName Storage_Tank_Multi_Inload, InstanceOfType FB
"Storage_Tank_Multi_Inload"
BEGIN
END_DATA_BLOCK

DATA_BLOCK "T-34.00"   // DB42
VERSION : 0.1
// stored: AutoNumber false, DBAccessibleFromOPCUA true, DBAccessibleFromWebserver true, InstanceOfName Storage_Tank_Multi_Inload, InstanceOfType FB
"Storage_Tank_Multi_Inload"
BEGIN
END_DATA_BLOCK

DATA_BLOCK "T-35.00"   // DB43
VERSION : 0.1
// stored: AutoNumber false, DBAccessibleFromOPCUA true, DBAccessibleFromWebserver true, InstanceOfName Storage_Tank_Multi_Inload, InstanceOfType FB
"Storage_Tank_Multi_Inload"
BEGIN
END_DATA_BLOCK

DATA_BLOCK "T-39.00"   // DB40
VERSION : 0.1
// stored: AutoNumber false, DBAccessibleFromOPCUA true, DBAccessibleFromWebserver true, InstanceOfName Storage_Tank_Single_Inload, InstanceOfType FB
"Storage_Tank_Single_Inload"
BEGIN
END_DATA_BLOCK

DATA_BLOCK "T-79.00"   // DB54
VERSION : 0.1
// stored: AutoNumber false, DBAccessibleFromOPCUA true, DBAccessibleFromWebserver true, InstanceOfName Storage_Tank_Multi_Inload, InstanceOfType FB
"Storage_Tank_Multi_Inload"
BEGIN
END_DATA_BLOCK

DATA_BLOCK "T-81.00"   // DB51
VERSION : 0.1
// stored: AutoNumber false, DBAccessibleFromOPCUA true, DBAccessibleFromWebserver true, InstanceOfName Storage_Tank_Multi_Inload, InstanceOfType FB
"Storage_Tank_Multi_Inload"
BEGIN
END_DATA_BLOCK

